// Return if no parameter is remaining...
IF ( ParameterCnt = 0 ) THEN RETURN; END_IF
// dec remaining parameter(s)                        
ParameterCnt := ParameterCnt - 1;
// Create log entry for HoldToRun
CreateLogMessagePara1 ( Timestamp   := AxesGroup.State.SystemTime,
                        MessageType := MessageType.CMD,
                        Severity    := Severity.DEBUG,
                        MessageCode := 0,
                        MessageText := 'Command.HoldToRun = {1}',
                        Para1       :=  BOOL_TO_STRING(_command.HoldToRun));
                        

// Return if no parameter is remaining...
IF ( ParameterCnt = 0 ) THEN RETURN; END_IF
// dec remaining parameter(s)                        
ParameterCnt := ParameterCnt - 1;
// Create log entry for StepMode
CreateLogMessagePara1 ( Timestamp   := AxesGroup.State.SystemTime,
                        MessageType := MessageType.CMD,
                        Severity    := Severity.DEBUG,
                        MessageCode := 0,
                        MessageText := 'Command.StepMode = {1}',
                        Para1       :=  USINT_TO_STRING(_command.StepMode));
                                                

// Return if no parameter is remaining...
IF ( ParameterCnt = 0 ) THEN RETURN; END_IF
// dec remaining parameter(s)                        
ParameterCnt := ParameterCnt - 1;
// Create log entry for ManualStep
CreateLogMessagePara1 ( Timestamp   := AxesGroup.State.SystemTime,
                        MessageType := MessageType.CMD,
                        Severity    := Severity.DEBUG,
                        MessageCode := 0,
                        MessageText := 'Command.ManualStep = {1}',
                        Para1       :=  BOOL_TO_STRING(_command.ManualStep));

                
END_METHOD

METHOD FB_init : BOOL
VAR_INPUT
  /// if TRUE, the retain variables are initialized (warm start / cold start)
  bInitRetains : BOOL; 
  /// if TRUE, the instance afterwards gets moved into the copy code (online change)
  bInCopyCode  : BOOL;  
END_VAR
                  MyType := 'MC_EnableRobotFB';

ExecMode := ExecutionMode.PARALLEL;
Priority := PriorityLevel.NORMAL;
                
END_METHOD

METHOD Protected OnExecCancel : DINT
VAR_IN_OUT
  /// Robot assignment of function
  AxesGroup : AxesGroup; 
END_VAR
VAR
  /// internal return value 
 _retVal    : DINT;
END_VAR
                  OnExecCancel := RobotLibraryConstants.RUNNING;

CASE _stepCancel OF
  
  0: // set busy flag
     Busy := TRUE;
    
     // Create log entry
     CreateLogMessagePara1 ( Timestamp   := AxesGroup.State.SystemTime,
                             MessageType := MessageType.CMD,
                             Severity    := Severity.DEBUG,
                             MessageCode := 0,
                             MessageText := 'Execution of {1} cancelled',
                             Para1       := MyType);                 
    
     // try to remove cmd
    _retVal := AxesGroup.Acyclic.ActiveCommandRegister.RemoveCmd(_uniqueID);
  
     // check result of removement       
     IF ( _retVal = RobotLibraryConstants.OK )
     THEN
       // Reset step counter
      _stepCancel := 0;
       // finished okay
       OnExecCancel := RobotLibraryConstants.OK;
     
       // Create log entry
       CreateLogMessagePara1 ( Timestamp   := AxesGroup.State.SystemTime,
                               MessageType := MessageType.CMD,
                               Severity    := Severity.DEBUG,
                               MessageCode := 0,
                               MessageText := '{1} successfully removed from ACR',
                               Para1       := MyType);                 
     ELSE
       // set timeout
       SetTimeout(PT := _timeoutCancel, rTimer := _timerCancel);
       // inc step counter
      _stepCancel := _stepCancel + 1; 
     
       // Create log entry
       CreateLogMessagePara1 ( Timestamp   := AxesGroup.State.SystemTime,
                               MessageType := MessageType.CMD,
                               Severity    := Severity.DEBUG,
                               MessageCode := 0,
                               MessageText := '{1} was not removed from ACR because execution was already in progress',
                               Para1       := MyType);                 
     END_IF       
  
     
 1:  // call clear error 
     OnExecCancel := OnExecErrorClear(AxesGroup := AxesGroup);  
 
     IF ( OnExecCancel = RobotLibraryConstants.OK)
     THEN
       // Reset busy flag
       Busy := FALSE;
       // Reset step counter
      _stepCancel := 0;
       // finished okay
       OnExecCancel := RobotLibraryConstants.OK;
     END_IF  
  
ELSE
  // invalid step
  SetError( ErrorID := RobotLibraryErrorIdEnum.ERR_INVALID_STEP, Overwrite := TRUE );
END_CASE  


                        
// reset step counter
IF (OnExecCancel <> RobotLibraryConstants.RUNNING)
THEN
  // Reset FB variables
  Reset();
  // Reset step counter
 _stepCancel := 0;
END_IF                        
                
END_METHOD

METHOD PROTECTED OnExecErrorClear : DINT
VAR_IN_OUT
  /// Robot assignment of function
  AxesGroup : AxesGroup; 
END_VAR
                  OnExecErrorClear := RobotLibraryConstants.RUNNING;

CASE _stepClearError OF
  
  0:  // set busy flag
      Busy := TRUE;
      // trigger parameter update to disable FB
     _parameterUpdateInternal := TRUE;
      // call Check Parameter changed method to trigger the parameter update to disable the function
      CheckParameterChanged(AxesGroup := AxesGroup);
      // set timeout
      SetTimeout(PT := _timeoutClearError, rTimer := _timerClearError);
      // inc step counter
     _stepClearError := _stepClearError + 1; 
      
  1: IF ( _responseReceived )
     THEN
       // reset response received flag
      _responseReceived := FALSE;
       // reset step counter
      _stepClearError := 0;
       // finished
       OnExecErrorClear := RobotLibraryConstants.OK;
     ELSE
       // timeout exceeded ? 
       IF (CheckTimeout(_timerClearError) = RobotLibraryConstants.OK)
       THEN
         OnExecErrorClear := RobotLibraryConstants.HAS_ERROR;
       END_IF
	   END_IF
ELSE
  // invalid step
  SetError( ErrorID := RobotLibraryErrorIdEnum.ERR_INVALID_STEP, Overwrite := TRUE );
END_CASE


// reset step counter
IF (OnExecErrorClear <> RobotLibraryConstants.RUNNING)
THEN
  // Reset 
  Reset();     
  // reset step counter
 _stepClearError := 0;
END_IF
                
END_METHOD

METHOD PROTECTED OnExecRun : DINT
VAR_IN_OUT
  /// Robot assignment of function
  AxesGroup : AxesGroup; 
END_VAR
                  SUPER^.OnExecRun(AxesGroup := AxesGroup);

CASE _stepCmd OF
  
  00:  IF ( _enable_R.Q ) AND ( NOT Error) 
       THEN
         // reset the rising edge
        _enable_R();       

         // Check function is supported and parameter are valid ?
         IF (( CheckFunctionSupported   ( AxesGroup := AxesGroup )) AND
             ( CheckParameterValid      ( AxesGroup := AxesGroup )) AND
             ( CheckSynchronizationValid( AxesGroup := AxesGroup )))      
         THEN
           // Reset all internal flags
           Reset();
           // set busy flag
           Busy := TRUE;
           // Reset command outputs
           SysDepMemSet(pDest := ADR(OutCmd), Value := 0, DataLen := SIZEOF(OutCmd));         
           // apply command parameter
          _parCmd := ParCmd;
           // init parameter sequence
          _command.ParSeq := 1;
           // create command data
           CommandData := CreateCommandPayload(AxesGroup := AxesGroup);
           // Add command to active command register
          _uniqueID := AxesGroup.Acyclic.ActiveCommandRegister.AddCmd( pCommandFB := ADR(THIS^ ));     
           // set timeout
           SetTimeout(PT := _timeoutCmd, rTimer := _timerCmd);
           // inc step counter
          _stepCmd := _stepCmd + 1; 
         END_IF
       END_IF
     

  01:  // Wait for responce received
       IF ( _responseReceived )
       THEN
         // reset response received flag
        _responseReceived := FALSE;
         // update state flags
         OnUpdateStateFlags(_response.State);
         // update state flags
         OnApplyOutCmd(_response.State);
       END_IF
       
       // do not abort directly, so that the ParSeq update can be send
       IF ( _enable_F.Q ) 
       THEN
         // Set Busy flag
         Busy := TRUE;
         // trigger parameter update to disable FB
        _parameterUpdateInternal := TRUE;        
         // reset the falling edge
        _enable_F();
         // set timeout
         SetTimeout(PT := _timeoutCmd, rTimer := _timerCmd);
         // inc step counter
        _stepCmd := _stepCmd + 1; 
       END_IF

      // Wait for response received or timeout or not Initialized
  02: IF ((    _responseReceived                                   )  OR 
          (     CheckTimeout(_timerCmd) = RobotLibraryConstants.OK )) OR 
         (( NOT AxesGroup.State.Initialized                        )  AND
          ( NOT AxesGroup.State.Synchronized                       ))
      THEN
        Reset();   
	    END_IF
      
ELSE
  // invalid step
  SetError( ErrorID := RobotLibraryErrorIdEnum.ERR_INVALID_STEP, Overwrite := TRUE );
END_CASE



// Reset FB
IF (( _enable_R.Q ) OR
    ( _enable_F.Q ))
THEN
  Reset();
END_IF
                
END_METHOD

METHOD PROTECTED OnUpdateStateFlags
VAR_INPUT
  /// Command message state
  State : CmdMessageState;
END_VAR
                  // Reset State flags
;

// Update results
Enabled := _response.Enabled;

CASE State OF

  // No operation or process is active
  CmdMessageState.EMPTY               :;
  // Created but not yet started
  CmdMessageState.CREATED             :;
  // Buffered and awaiting execution
  CmdMessageState.BUFFERED            : CommandBuffered    := TRUE;
                                        ParameterAccepted  := TRUE;  
  // Buffered in planner for future execution
  CmdMessageState.BUFFERED_IN_PLANNER : CommandBuffered    := TRUE;
                                        ParameterAccepted  := TRUE;
  // Currently active and in progress
  CmdMessageState.ACTIVE              : IF (Enabled = Enable)
                                        THEN  
                                          Busy := FALSE;   
                                        END_IF
                                       
  // Interrupted and awaiting continuation
  CmdMessageState.INTERRUPTED         :;  
  // Requested for abort
  CmdMessageState.ABORT_REQUEST       :;
  // Successfully completed
  CmdMessageState.DONE                : Busy               := FALSE;
  // Aborted before completion
  CmdMessageState.ABORTED             : Busy               := FALSE;
  // Encountered an error during execution
  CmdMessageState.ERROR               : Error              := TRUE;
                                        Busy               := FALSE;
END_CASE
                
END_METHOD

METHOD INTERNAL ParseResponsePayload : DINT
VAR_INPUT
  /// Response data
  ResponseData : RobotLibraryResponseDataFB;
  /// Timestamp
  Timestamp    : SystemTime;  
END_VAR
VAR
  /// Parameter count
 _parameterCnt : DINT;
END_VAR
// Table 6-26: Received CMD payload (RC to PLC) of "EnableRobot"
// --------------------------
// Header
// --------------------------
// Byte 00 : USINT - ParSeq | State     
// Byte 01 : SINT  - AlarmMessageSeverity    
// Byte 02 : UINT  - AlarmMessageCode HB
// Byte 03 :       - AlarmMessageCode LB
// --------------------------
// Datablock
// --------------------------
// Byte 04 : BOOL  - Enabled
// --------------------------
                  // call base implementation to parse the header from payload buffer
ResponseData.PayloadPtr := SUPER^.ParseResponsePayload(ResponseData := ResponseData, Timestamp := Timestamp);

// copy parsed header to response
_response.ParSeq               := _rspHeader.ParSeq;
_response.State                := _rspHeader.State;
_response.AlarmMessageSeverity := _rspHeader.AlarmMessageSeverity;
_response.AlarmMessageCode     := _rspHeader.AlarmMessageCode;


// Check payload remaining ? 
IF ( ResponseData.IsPayloadRemaining)
THEN 
  // Get Response.Enabled
 _response.Enabled := ResponseData.GetBool();
  // inc parameter counter
 _parameterCnt := _parameterCnt + 1;
END_IF


// Create logging
ParseResponsePayloadLog(ResponseData := ResponseData, Timestamp := Timestamp, ParameterCnt := _parameterCnt);
                
END_METHOD

METHOD INTERNAL ParseResponsePayloadLog
VAR_INPUT
  /// Response data
  ResponseData : RobotLibraryResponseDataFB;
  /// Timestamp
  Timestamp    : SystemTime;  
  /// Parameter count
  ParameterCnt : DINT;
END_VAR
                  // Create log entry for Parameter start
CreateLogMessagePara1 ( Timestamp   := Timestamp,
                        MessageType := MessageType.CMD,
                        Severity    := Severity.DEBUG,
                        MessageCode := 0,
                        MessageText := '{1} parameter(s) to parse from the response data:',
                        Para1       := DINT_TO_STRING(ParameterCnt));
                        
// Return if no parameter is remaining...
IF ( ParameterCnt = 0 ) THEN RETURN; END_IF
// dec remaining parameter(s)                        
ParameterCnt := ParameterCnt - 1;

// Create log entry for Enabled
CreateLogMessagePara1 ( Timestamp   := Timestamp,
                        MessageType := MessageType.CMD,
                        Severity    := Severity.DEBUG,
                        MessageCode := 0,
                        MessageText := 'Response.Enabled = {1}',
                        Para1       :=  BOOL_TO_STRING(_response.Enabled));


                
END_METHOD

METHOD PROTECTED Reset : DINT
VAR_INPUT
END_VAR
                  SUPER^.Reset();

Busy               := FALSE;
CommandBuffered    := FALSE;
ParameterAccepted  := FALSE;
                
END_METHOD
END_FUNCTION_BLOCK

/// Acknowledgement all pending errors
FUNCTION_BLOCK MC_GroupResetFB EXTENDS RobotLibraryBaseExecuteFB
// ------------------------------------------------------------------------- 
//  SRCI Robot Library                                                
// ------------------------------------------------------------------------- 
//                                                                           
//  Object:      GroupResetFB                                       
//  Author:      Thorsten Brach                                                
//  Date:        2024-06-01
//
//  Description:                                              
//   
//                                                                           
//  Copyright: 
//    (C) 2024 Thorsten Brach. All rights reserved                                                                                                                                            
//             Licensed under the MIT License.
//                                                                           
//  Disclaimer:                                                                           
//    This project is provided without any guarantee and can be used for   
//    private and commercial purposes. Any use is at the user’s 
//    own risk and responsibility.
//
// -------------------------------------------------------------------------
VAR_INPUT
  /// Command parameter 
  ParCmd          : GroupResetParCmd;      
END_VAR

VAR_OUTPUT
  /// Command output 
  OutCmd          : GroupResetOutCmd;   
  /// Command is transferred and confirmed by the RC
  CommandBuffered : BOOL;     
END_VAR
VAR
  /// internal copy of command parameter 
 _parCmd          : GroupResetParCmd;
  /// command data to send
 _command         : GroupResetSendData;
  /// response data received
 _response        : GroupResetRecvData;      
END_VAR

            SUPER^(AxesGroup := AxesGroup);
          

METHOD INTERNAL CheckAddParameter : BOOL
VAR_INPUT
  /// Payload pointer
  PayloadPtr : UDINT;
END_VAR
VAR
  /// Payload as byte array
  Payload    : ARRAY [1..SIZEOF(_command)] OF BYTE;
  /// Null Byte array 
  Null       : ARRAY [1..SIZEOF(_command)] OF BYTE;
  /// Data length to compare
  DataLen    : UDINT;
END_VAR
                  // Payload pointer must be decreased by one byte, because ADR(Payload) is already one byte !
PayloadPtr := LIMIT (0, PayloadPtr - 1, SIZEOF(Payload) -1);
// Convert command struct to payload array
SysDepMemCpy( pDest := ADR(Payload), pSrc := ADR(_command), DataLen := SIZEOF(_command));
// Calculate the data length to compare - at least one byte must be compared !
DataLen := LIMIT(1, SIZEOF(Payload) - PayloadPtr, SIZEOF(Payload)); 
// Compare Payload-Array with Null-Byte-Array
CheckAddParameter := SysDepMemCmp( pData1 := ADR(Payload) + PayloadPtr , pData2 := ADR(Null), DataLen := DataLen) <>  RobotLibraryConstants.OK ;
                
END_METHOD

METHOD PROTECTED CheckFunctionSupported : BOOL
VAR_IN_OUT
  /// Robot assignment of function
  AxesGroup : AxesGroup; 
END_VAR
                  CheckFunctionSupported := AxesGroup.State.RobotData.RCSupportedFunctions.GroupReset;

IF ( NOT CheckFunctionSupported )
THEN
  // call base implementation for set error and create log entry
  SUPER^.CheckFunctionSupported(AxesGroup := AxesGroup);
END_IF
                
END_METHOD

METHOD PROTECTED CheckParameterChanged : BOOL
VAR_IN_OUT
  /// Robot assignment of function
  AxesGroup    : AxesGroup; 
END_VAR
                  IF (SIZEOF(ParCmd) = 0) OR (_stepCmd = 0)
THEN
  RETURN;
END_IF
 
// compare memory
_parameterChanged := ( SysDepMemCmp(pData1 := ADR(ParCmd), pData2 := ADR(_parCmd), DataLen := SIZEOF(ParCmd)) <> RobotLibraryConstants.OK );

// check parameter valid ?
_parameterValid   := CheckParameterValid( AxesGroup := AxesGroup );

IF ((  _parameterChanged        )  AND 
    (  _parameterValid          )) OR
    (  _parameterUpdateInternal )  
THEN  
  // Create log entry for parameter changed event
  CreateLogMessagePara1 ( Timestamp   := AxesGroup.State.SystemTime,
                          MessageType := MessageType.CMD,
                          Severity    := Severity.DEBUG,
                          MessageCode := 0,
                          MessageText := 'NotifyParameterChanged Event {1}',
                          Para1       :=  '' );

  // reset internal flag for send parameter update
 _parameterUpdateInternal := FALSE;
  // update internal copy of parameters 
 _parCmd := ParCmd;
  // inc parameter sequence
 _command.ParSeq := _command.ParSeq + 1;
  // update command data  
  CommandData := CreateCommandPayload(AxesGroup := AxesGroup); // ( Access via reference to rCommandFB in ACR )
  // notify active command register 
  AxesGroup.Acyclic.ActiveCommandRegister.NotifyParameterChanged := _uniqueID;
END_IF
                
END_METHOD

METHOD INTERNAL CreateCommandPayload : RobotLibraryCommandDataFB
VAR_IN_OUT
  /// Robot assignment of function
  AxesGroup : AxesGroup; 
END_VAR
VAR
  /// Parameter count
 _parameterCnt : DINT;
END_VAR
// Table 6-31: Sent CMD payload (PLC to RC) of "GroupReset"
// --------------------------
// Header
// --------------------------
// Byte 00 : UINT  - Type HB     
// Byte 01 :       - Type LB    
// Byte 02 : USINT - Reserve | ExecutionMode
// Byte 03 : USINT - ParSeq  | Priority
// --------------------------
                  // set command parameter 
_command.CmdTyp     :=  CmdType.GroupReset;
_command.ExecMode   :=  ExecMode;
_command.ParSeq     := _command.ParSeq;
_command.Priority   :=  Priority;

// copy command data to header
_cmdHeader := _command;
// call base implementation to copy header to payload buffer
CreateCommandPayload := SUPER^.CreateCommandPayload(AxesGroup := AxesGroup);


// Create logging
CreateCommandPayloadLog(AxesGroup := AxesGroup, ParameterCnt := _parameterCnt);
                
END_METHOD

METHOD INTERNAL CreateCommandPayloadLog
VAR_IN_OUT
  /// Robot assignment of function
  AxesGroup : AxesGroup; 
END_VAR
VAR_INPUT
  /// Parameter count
  ParameterCnt : DINT;
END_VAR
                  // Create log entry for Parameter start
CreateLogMessagePara1 ( Timestamp   := AxesGroup.State.SystemTime,
                        MessageType := MessageType.CMD,
                        Severity    := Severity.DEBUG,
                        MessageCode := 0,
                        MessageText := 'Create command payload with {1} parameter(s) :',
                        Para1       := DINT_TO_STRING(ParameterCnt));
                
END_METHOD

METHOD FB_init : BOOL
VAR_INPUT
  /// if TRUE, the retain variables are initialized (warm start / cold start)
  bInitRetains : BOOL; 
  /// if TRUE, the instance afterwards gets moved into the copy code (online change)
  bInCopyCode  : BOOL;  
END_VAR
                  MyType := 'MC_GroupResetFB';

ExecMode := ExecutionMode.PARALLEL;
Priority := PriorityLevel.NORMAL;
                
END_METHOD

METHOD PROTECTED OnExecRun : DINT
VAR_IN_OUT
  /// Robot assignment of function
  AxesGroup : AxesGroup; 
END_VAR
                  // call base implementation
SUPER^.OnExecRun(AxesGroup := AxesGroup);

CASE _stepCmd OF
  
  00:  IF ( _execute_R.Q ) AND ( NOT Error)
       THEN
         IF (( CheckFunctionSupported( AxesGroup := AxesGroup )) AND
             ( CheckParameterValid   ( AxesGroup := AxesGroup )))      
         THEN
           // set busy flag
           Busy := TRUE;
           // Reset command outputs
           SysDepMemSet(pDest := ADR(OutCmd), Value := 0, DataLen := SIZEOF(OutCmd));         
           // apply command parameter
          _parCmd := ParCmd;
           // init parameter sequence
          _command.ParSeq := 1;
           // create command data
           CommandData := CreateCommandPayload(AxesGroup := AxesGroup);
           // Add command to active command register
          _uniqueID := AxesGroup.Acyclic.ActiveCommandRegister.AddCmd( pCommandFB := ADR(THIS^ ));     
           // set timeout
           SetTimeout(PT := _timeoutCmd, rTimer := _timerCmd);
           // inc step counter
          _stepCmd := _stepCmd + 1;
         END_IF 
       END_IF
     

  01:  // Wait for responce received
       IF ( _responseReceived )
       THEN
         // reset response received flag
        _responseReceived := FALSE;
         // update state flags
         OnUpdateStateFlags(_response.State);
         // update state flags
         OnApplyOutCmd(_response.State);
               
         // Done, Aborted or Error ?
         IF (_response.State >= CmdMessageState.DONE )
         THEN
           // Reset FastStop counter
           AxesGroup.Cyclic.PlcToRob.FastStop := 0; 
           // set timeout
           SetTimeout(PT := _timeoutCmd, rTimer := _timerCmd);
           // inc step counter
          _stepCmd := _stepCmd + 1; 
         END_IF
       END_IF


  02: IF ( NOT Execute)
      THEN
        Reset();
      END_IF     

ELSE
  // invalid step
  SetError( ErrorID := RobotLibraryErrorIdEnum.ERR_INVALID_STEP, Overwrite := TRUE );
END_CASE


// Reset FB
IF ( NOT Execute )
THEN
  Reset();
END_IF

// forwarding GroupReset Info
AxesGroup.State.GroupReset := Execute;
                
END_METHOD

METHOD PROTECTED OnUpdateStateFlags
VAR_INPUT
  /// Command message state
  State : CmdMessageState;
END_VAR
                  // Reset State flags
Done := FALSE;

CASE State OF

  // No operation or process is active
  CmdMessageState.EMPTY               :;
  // Created but not yet started
  CmdMessageState.CREATED             :;
  // Buffered and awaiting execution
  CmdMessageState.BUFFERED            : CommandBuffered    := TRUE;
  // Buffered in planner for future execution
  CmdMessageState.BUFFERED_IN_PLANNER : CommandBuffered    := TRUE;
  // Currently active and in progress
  CmdMessageState.ACTIVE              :;                                         
  // Interrupted and awaiting continuation
  CmdMessageState.INTERRUPTED         :;  
  // Requested for abort
  CmdMessageState.ABORT_REQUEST       :;
  // Successfully completed
  CmdMessageState.DONE                : Done               := TRUE;
                                        Busy               := FALSE;
  // Aborted before completion
  CmdMessageState.ABORTED             : Busy               := FALSE;
  // Encountered an error during execution
  CmdMessageState.ERROR               : Error              := TRUE;
                                        Busy               := FALSE;
END_CASE
                
END_METHOD

METHOD INTERNAL ParseResponsePayload : DINT
VAR_INPUT
  /// Response data
  ResponseData : RobotLibraryResponseDataFB;
  /// Timestamp
  Timestamp    : SystemTime;  
END_VAR
VAR
  /// Parameter count
 _parameterCnt : DINT;
END_VAR
// Table 6-32: Received CMD payload (RC to PLC) of "GroupReset"
// --------------------------
// Header
// --------------------------
// Byte 00 : USINT - ParSeq | State     
// Byte 01 : SINT  - AlarmMessageSeverity    
// Byte 02 : UINT  - AlarmMessageCode HB
// Byte 03 :       - AlarmMessageCode LB
                  // call base implementation to parse the header from payload buffer
ResponseData.PayloadPtr := SUPER^.ParseResponsePayload(ResponseData := ResponseData, Timestamp := Timestamp);

// copy parsed header to response
_response.ParSeq               := _rspHeader.ParSeq;
_response.State                := _rspHeader.State;
_response.AlarmMessageSeverity := _rspHeader.AlarmMessageSeverity;
_response.AlarmMessageCode     := _rspHeader.AlarmMessageCode;

// Create logging
ParseResponsePayloadLog(ResponseData := ResponseData, Timestamp := Timestamp, ParameterCnt := _parameterCnt);
                
END_METHOD

METHOD INTERNAL ParseResponsePayloadLog
VAR_INPUT
  /// Response data
  ResponseData : RobotLibraryResponseDataFB;
  /// Timestamp
  Timestamp    : SystemTime;  
  /// Parameter count
  ParameterCnt : DINT;
END_VAR
                  // Create log entry for Parameter start
CreateLogMessagePara1 ( Timestamp   := Timestamp,
                        MessageType := MessageType.CMD,
                        Severity    := Severity.DEBUG,
                        MessageCode := 0,
                        MessageText := '{1} parameter(s) to parse from the response data:',
                        Para1       := DINT_TO_STRING(ParameterCnt));
                        

// Return if no parameter is remaining...
IF ( ParameterCnt = 0 ) THEN RETURN; END_IF
// dec remaining parameter(s)                        
ParameterCnt := ParameterCnt - 1;
// Create log entry for no parameter 
CreateLogMessage      ( Timestamp   := Timestamp,
                        MessageType := MessageType.CMD,
                        Severity    := Severity.DEBUG,
                        MessageCode := 0,
                        MessageText := 'This command has no parameter to parse...');
                
END_METHOD

METHOD PROTECTED Reset : DINT
VAR_INPUT
END_VAR
                  Reset := SUPER^.Reset();

Done               := FALSE;
Busy               := FALSE;
CommandBuffered    := FALSE;


                
END_METHOD
END_FUNCTION_BLOCK

FUNCTION_BLOCK MC_ReadServerLog EXTENDS RobotLibraryBaseFB
VAR
END_VAR

            
          

METHOD FB_init : BOOL
VAR_INPUT
  /// if TRUE, the retain variables are initialized (warm start / cold start)
  bInitRetains : BOOL; 
  /// if TRUE, the instance afterwards gets moved into the copy code (online change)
  bInCopyCode  : BOOL;  
END_VAR
                  MyType := 'MC_ReadServerLogFB';

ExecMode := ExecutionMode.PARALLEL;
Priority := PriorityLevel.NORMAL;
                
END_METHOD
END_FUNCTION_BLOCK

/// Restart/reboot of the RC.
FUNCTION_BLOCK MC_RestartControllerFB EXTENDS RobotLibraryBaseExecuteFB
// ------------------------------------------------------------------------- 
//  SRCI Robot Library                                                
// ------------------------------------------------------------------------- 
//                                                                           
//  Object:      RestartControllerFB                                       
//  Author:      Thorsten Brach                                                
//  Date:        2024-06-01
//
//  Description:                                              
//   
//                                                                           
//  Copyright: 
//    (C) 2024 Thorsten Brach. All rights reserved                                                                                                                                            
//             Licensed under the MIT License.
//                                                                           
//  Disclaimer:                                                                           
//    This project is provided without any guarantee and can be used for   
//    private and commercial purposes. Any use is at the user’s 
//    own risk and responsibility.
//
// -------------------------------------------------------------------------
VAR_INPUT
  /// Command parameter 
  ParCmd          : RestartControllerParCmd;  
END_VAR

VAR_OUTPUT
  /// Command is transferred and confirmed by the RC
  CommandBuffered : BOOL;
  /// Command outputs 
  OutCmd          : RestartControllerOutCmd;  
END_VAR

VAR
  /// internal copy of command parameter 
 _parCmd          : RestartControllerParCmd;
  /// command data to send
 _command         : RestartControllerSendData;
  /// response data received
 _response        : RestartControllerRecvData;      
END_VAR

            SUPER^(AxesGroup := AxesGroup);
          

METHOD INTERNAL CheckAddParameter : BOOL
VAR_INPUT
  /// Payload pointer
  PayloadPtr : UDINT;
END_VAR
VAR
  /// Payload as byte array
  Payload    : ARRAY [1..SIZEOF(_command)] OF BYTE;
  /// Null Byte array 
  Null       : ARRAY [1..SIZEOF(_command)] OF BYTE;
  /// Data length to compare
  DataLen    : UDINT;
END_VAR
                  // Payload pointer must be decreased by one byte, because ADR(Payload) is already one byte !
PayloadPtr := LIMIT (0, PayloadPtr - 1, SIZEOF(Payload) -1);
// Convert command struct to payload array
SysDepMemCpy( pDest := ADR(Payload), pSrc := ADR(_command), DataLen := SIZEOF(_command));
// Calculate the data length to compare - at least one byte must be compared !
DataLen := LIMIT(1, SIZEOF(Payload) - PayloadPtr, SIZEOF(Payload)); 
// Compare Payload-Array with Null-Byte-Array
CheckAddParameter := SysDepMemCmp( pData1 := ADR(Payload) + PayloadPtr , pData2 := ADR(Null), DataLen := DataLen) <>  RobotLibraryConstants.OK ;
                
END_METHOD

METHOD PROTECTED CheckFunctionSupported : BOOL
VAR_IN_OUT
  /// Robot assignment of function
  AxesGroup : AxesGroup; 
END_VAR
                  CheckFunctionSupported := AxesGroup.State.RobotData.RCSupportedFunctions.RestartController;

IF ( NOT CheckFunctionSupported )
THEN
  // call base implementation for set error and create log entry
  SUPER^.CheckFunctionSupported(AxesGroup := AxesGroup);
END_IF
                
END_METHOD

METHOD PROTECTED CheckParameterChanged : BOOL
VAR_IN_OUT
  /// Robot assignment of function
  AxesGroup    : AxesGroup; 
END_VAR
                  // Check ParCmd Size is > 0, because MemCmp does not work correctly with size = 0
IF (SIZEOF(ParCmd) = 0) OR (_stepCmd = 0)
THEN 
  RETURN;
END_IF

// compare memory 
_parameterChanged := ( SysDepMemCmp(pData1 := ADR(ParCmd), pData2 := ADR(_parCmd), DataLen := SIZEOF(ParCmd)) <> RobotLibraryConstants.OK );

// check parameter valid ?
_parameterValid   := CheckParameterValid( AxesGroup := AxesGroup );

IF ((  _parameterChanged        )  AND 
    (  _parameterValid          )) OR
    (  _parameterUpdateInternal )  
THEN  
  // Create log entry for parameter changed event
  CreateLogMessagePara1 ( Timestamp   := AxesGroup.State.SystemTime,
                          MessageType := MessageType.CMD,
                          Severity    := Severity.DEBUG,
                          MessageCode := 0,
                          MessageText := 'NotifyParameterChanged Event {1}',
                          Para1       :=  '' );

  // reset internal flag for send parameter update
 _parameterUpdateInternal := FALSE;
  // update internal copy of parameters 
 _parCmd := ParCmd;
  // inc parameter sequence
 _command.ParSeq := _command.ParSeq + 1;
  // update command data  
  CommandData := CreateCommandPayload(AxesGroup := AxesGroup); // ( Access via reference to rCommandFB in ACR )
  // notify active command register 
  AxesGroup.Acyclic.ActiveCommandRegister.NotifyParameterChanged := _uniqueID;
END_IF
                
END_METHOD

METHOD INTERNAL CreateCommandPayload : RobotLibraryCommandDataFB
VAR_IN_OUT
  /// Robot assignment of function
  AxesGroup : AxesGroup; 
END_VAR
VAR
  /// Parameter count
 _parameterCnt : DINT;
END_VAR
// Table 6-57: Sent CMD payload (PLC to RC) of "RestartController"
// --------------------------
// Header
// --------------------------
// Byte 00 : UINT  - Type HB     
// Byte 01 :       - Type LB    
// Byte 02 : USINT - Reserve | ExecutionMode
// Byte 03 : USINT - ParSeq  | Priority
// --------------------------
                  // set command parameter 
_command.CmdTyp     :=  CmdType.RestartController;
_command.ExecMode   :=  ExecMode;
_command.ParSeq     := _command.ParSeq;
_command.Priority   :=  Priority;


// copy command data to header
_cmdHeader := _command;
// call base implementation to copy header to payload buffer
CreateCommandPayload := SUPER^.CreateCommandPayload(AxesGroup := AxesGroup);


// Create logging
CreateCommandPayloadLog(AxesGroup := AxesGroup, ParameterCnt := _parameterCnt);
                
END_METHOD

METHOD INTERNAL CreateCommandPayloadLog
VAR_IN_OUT
  /// Robot assignment of function
  AxesGroup : AxesGroup; 
END_VAR
VAR_INPUT
  /// Parameter count
  ParameterCnt : DINT;
END_VAR
                  // Create log entry for Parameter start
CreateLogMessagePara1 ( Timestamp   := AxesGroup.State.SystemTime,
                        MessageType := MessageType.CMD,
                        Severity    := Severity.DEBUG,
                        MessageCode := 0,
                        MessageText := 'Create command payload with {1} parameter(s) :',
                        Para1       := DINT_TO_STRING(ParameterCnt));
                
END_METHOD

METHOD FB_init : BOOL
VAR_INPUT
  /// if TRUE, the retain variables are initialized (warm start / cold start)
  bInitRetains : BOOL; 
  /// if TRUE, the instance afterwards gets moved into the copy code (online change)
  bInCopyCode  : BOOL;  
END_VAR
                  MyType := 'MC_RestartControllerFB';

ExecMode := ExecutionMode.PARALLEL;
Priority := PriorityLevel.NORMAL;
                
END_METHOD

METHOD PROTECTED OnApplyOutCmd
VAR_INPUT
  /// Command message state
  State : CmdMessageState;
END_VAR
                  IF ( State = CmdMessageState.EMPTY ) 
THEN
  // Reset command outputs
  SysDepMemSet(pDest := ADR(OutCmd), Value := 0, DataLen := SIZEOF(OutCmd));         
END_IF

IF (( State = CmdMessageState.ACTIVE ) OR
    ( State = CmdMessageState.DONE   ))
THEN
  // Update results
  OutCmd.RestartAccepted := _response.RestartAccepted;
END_IF
                
END_METHOD

METHOD PROTECTED OnExecRun : DINT
VAR_IN_OUT
  /// Robot assignment of function
  AxesGroup : AxesGroup; 
END_VAR
                  // call base implementation
SUPER^.OnExecRun(AxesGroup := AxesGroup);

CASE _stepCmd OF
  
  00:  IF ( _execute_R.Q ) AND ( NOT Error)   
       THEN
         // Check function is supported and parameter are valid ?
         IF (( CheckFunctionSupported( AxesGroup := AxesGroup )) AND
             ( CheckParameterValid   ( AxesGroup := AxesGroup )))      
         THEN
           // set busy flag
           Busy := TRUE;
           // Reset command outputs
           SysDepMemSet(pDest := ADR(OutCmd), Value := 0, DataLen := SIZEOF(OutCmd));         
           // apply command parameter
          _parCmd := ParCmd;
           // init parameter sequence
          _command.ParSeq := 1;
           // create command data
           CommandData := CreateCommandPayload(AxesGroup := AxesGroup);
           // Add command to active command register
          _uniqueID := AxesGroup.Acyclic.ActiveCommandRegister.AddCmd( pCommandFB := ADR(THIS^ ));     
           // set timeout
           SetTimeout(PT := _timeoutCmd, rTimer := _timerCmd);
           // inc step counter
          _stepCmd := _stepCmd + 1;
         END_IF 
       END_IF
     

  01:  // Wait for responce received
       IF ( _responseReceived )
       THEN
         // reset response received flag
        _responseReceived := FALSE;
         // update state flags
         OnUpdateStateFlags(_response.State);
         // update state flags
         OnApplyOutCmd(_response.State);

         // Done, Aborted or Error ?
         IF (_response.State >= CmdMessageState.DONE )
         THEN
           // set timeout
           SetTimeout(PT := _timeoutCmd, rTimer := _timerCmd);
           // inc step counter
          _stepCmd := _stepCmd + 1; 
         END_IF
       END_IF


  02: IF ( NOT Execute)
      THEN
        Reset();
      END_IF     

ELSE
  // invalid step
  SetError( ErrorID := RobotLibraryErrorIdEnum.ERR_INVALID_STEP, Overwrite := TRUE );
END_CASE


// Reset FB
IF ( NOT Execute )
THEN
  Reset();
END_IF
                
END_METHOD

METHOD PROTECTED OnUpdateStateFlags
VAR_INPUT
  /// Command message state
  State : CmdMessageState;
END_VAR
                  // Reset State flags
Done := FALSE;

CASE State OF

  // No operation or process is active
  CmdMessageState.EMPTY               :;
  // Created but not yet started
  CmdMessageState.CREATED             :;
  // Buffered and awaiting execution
  CmdMessageState.BUFFERED            : CommandBuffered    := TRUE;
  // Buffered in planner for future execution
  CmdMessageState.BUFFERED_IN_PLANNER : CommandBuffered    := TRUE;
  // Currently active and in progress
  CmdMessageState.ACTIVE              :;
  // Interrupted and awaiting continuation
  CmdMessageState.INTERRUPTED         :;  
  // Requested for abort
  CmdMessageState.ABORT_REQUEST       :;
  // Successfully completed
  CmdMessageState.DONE                : Done               := TRUE;
                                        Busy               := FALSE;
  // Aborted before completion
  CmdMessageState.ABORTED             : Busy               := FALSE;
  // Encountered an error during execution
  CmdMessageState.ERROR               : Error              := TRUE;
                                        Busy               := FALSE;
END_CASE
                
END_METHOD

METHOD INTERNAL ParseResponsePayload : DINT
VAR_INPUT
  /// Response data
  ResponseData : RobotLibraryResponseDataFB;
  /// Timestamp
  Timestamp    : SystemTime;  
END_VAR
VAR
  /// Parameter count
 _parameterCnt : DINT;
END_VAR
// Table 6-58: Received CMD payload (RC to PLC) of "RestartController"
// --------------------------
// Header
// --------------------------
// Byte 00 : USINT - ParSeq | State     
// Byte 01 : SINT  - AlarmMessageSeverity    
// Byte 02 : UINT  - AlarmMessageCode HB
// Byte 03 :       - AlarmMessageCode LB
// --------------------------
// Datablock
// --------------------------
// Byte 4  : BOOL  - RestartAccepted
                  // call base implementation to parse the header from payload buffer
ResponseData.PayloadPtr := SUPER^.ParseResponsePayload(ResponseData := ResponseData, Timestamp := Timestamp);

// copy parsed header to response
_response.ParSeq               := _rspHeader.ParSeq;
_response.State                := _rspHeader.State;
_response.AlarmMessageSeverity := _rspHeader.AlarmMessageSeverity;
_response.AlarmMessageCode     := _rspHeader.AlarmMessageCode;

// Check payload remaining ? 
IF ( ResponseData.IsPayloadRemaining)
THEN 
  // Get Response.RestartAccepted
 _response.RestartAccepted := ResponseData.GetBool();
  // inc parameter counter
 _parameterCnt := _parameterCnt + 1;
END_IF


// Create logging
ParseResponsePayloadLog(ResponseData := ResponseData, Timestamp := Timestamp, ParameterCnt := _parameterCnt);
                
END_METHOD

METHOD INTERNAL ParseResponsePayloadLog
VAR_INPUT
  /// Response data
  ResponseData : RobotLibraryResponseDataFB;
  /// Timestamp
  Timestamp    : SystemTime;  
  /// Parameter count
  ParameterCnt : DINT;
END_VAR
                  // Create log entry for Parameter start
CreateLogMessagePara1 ( Timestamp   := Timestamp,
                        MessageType := MessageType.CMD,
                        Severity    := Severity.DEBUG,
                        MessageCode := 0,
                        MessageText := '{1} parameter(s) to parse from the response data:',
                        Para1       := DINT_TO_STRING(ParameterCnt));
                        

// Return if no parameter is remaining...
IF ( ParameterCnt = 0 ) THEN RETURN; END_IF
// dec remaining parameter(s)                        
ParameterCnt := ParameterCnt - 1;
// Create log entry for RestartAccepted
CreateLogMessagePara1 ( Timestamp   := Timestamp,
                        MessageType := MessageType.CMD,
                        Severity    := Severity.DEBUG,
                        MessageCode := 0,
                        MessageText := 'Response.RestartAccepted = {1}',
                        Para1       :=  BOOL_TO_STRING(_response.RestartAccepted));


                
END_METHOD

METHOD PROTECTED Reset : DINT
VAR_INPUT
END_VAR
                  Reset := SUPER^.Reset();

Done               := FALSE;
Busy               := FALSE;
CommandBuffered    := FALSE;

                
END_METHOD
END_FUNCTION_BLOCK

/// Handles multiple mechanisms required for operation of the interface.
/// For maximal performance, this FB must be called after the function FB's, 
/// so that the data can be written to the fieldbus in the same cycle as the start of FB occours 
FUNCTION_BLOCK MC_RobotTaskFB EXTENDS RobotLibraryLogFB
// ------------------------------------------------------------------------- 
//  SRCI Robot Library                                                
// ------------------------------------------------------------------------- 
//                                                                           
//  Object:      RobotTaskFB                                       
//  Author:      Thorsten Brach                                                
//  Date:        2024-06-01
//
//  Description:                                              
//   
//                                                                           
//  Copyright: 
//    (C) 2024 Thorsten Brach. All rights reserved                                                                                                                                            
//             Licensed under the MIT License.
//                                                                           
//  Disclaimer:                                                                           
//    This project is provided without any guarantee and can be used for   
//    private and commercial purposes. Any use is at the user’s 
//    own risk and responsibility.
//
// -------------------------------------------------------------------------
VAR_INPUT
  /// Set TRUE (default) to initialize the interface
  Enable            : BOOL;
  /// User defined robot name
  RobotName         : STRING(20);
  /// Current System Time
  SystemTime        : SystemTime;
  /// Online Change detected
  OnlineChange      : BOOL;
  /// Axes Group ID -> is used to uniquely identify each RA on a per RC basis.
  ///
  /// For convenience, an RC with only one RA must assign ID 1 to this RA. 
  /// An RC with multiple RAs must assign numeric values 1-15 to those RAs.
  AxesGroupID       : BYTE := 0; // ToDo: Mistake in specification : ID should start with 1, but must start with 0 !  
  /// Configuration parameter
  ParCfg            : RobotTaskParCfg;
END_VAR

VAR_IN_OUT
  /// Inputs of PLC for communication from RC
  RobotInData       : ARRAY[*] OF BYTE;
  /// Outputs of PLC for communication to RC
  RobotOutData      : ARRAY[*] OF BYTE;
  ///  User data stored on the PLC according to Table 6-10
  UserData          : UserData;
  /// ToolData stored on PLC. For more information refer to 5.5.6.3
  ToolData          : ARRAY[*] OF Tool;
  /// LoadData stored on PLC.For more information refer to 5.5.6.4
  FrameData         : ARRAY[*] OF Frame;
  /// LoadData stored on PLC.For more information refer to 5.5.6.4 
  LoadData          : ARRAY[*] OF Load;
  /// Work areas stored on PLC. For more information refer to 5.5.8
  WorkAreas         : ARRAY[*] OF RobotWorkArea;
  /// Software limits stored on PLC
  SWLimits          : SWLimits;
  /// Default dynamics stored on PLC. For more information refer to 5.5.7
  DefaultDynamics   : DefaultDynamics;
  /// Reference dynamics stored on PLC. For more information refer to 5.5.7
  ReferenceDynamics : ReferenceDynamics;
  /// System log on PLC
  SystemLog         : ARRAY[0..RobotLibraryParameter.SYSTEM_LOG_MAX ] OF STRING(RobotLibraryParameter.MESSAGE_TEXT_LEN);
  /// Message buffer on the PLC - For more information refer to 5.5.11
  MessageLog        : ARRAY[0..RobotLibraryParameter.MESSAGE_LOG_MAX] OF AlarmMessage;
  /// Robot assignment of function
  AxesGroup         : AxesGroup;
END_VAR

VAR_OUTPUT
  /// FB is being processed
  Busy              : BOOL;
  /// Interface is initialized (RI state: "Initialized").
  /// For more information on RI states refer to chapter 5.5.3.1.
  Initialized       : BOOL;
  /// Server and client were successfully synchronized (RI state: "Synchronized").
  /// For more information on the synchronization mechanism refer to chapter 5.6.7.
  Synchronized      : BOOL;
  /// An error occurred
  Error             : BOOL;
  /// ErrorID reported by RC for error identification according to Table 7-1
  ErrorID           : WORD;
  ErrorIdEnum       : RobotLibraryErrorIdEnum;  
  ErrorAddTxt       : STRING(RobotLibraryConstants.MAX_ADD_TEXT_LENGTH);
  /// WarningID for warning identification reported during execution of command according to Table 7-3
  WarningID         : WORD;
  WarningIdEnum     : RobotLibraryWarningIdEnum;  
  /// InfoID for info identification reported during execution of command according to Table 7-5
  InfoID            : WORD;    
  InfoIdEnum        : RobotLibraryInfoIdEnum;    
END_VAR

VAR
  /// internal copy of configuration parameter
 _parCfg                       : RobotTaskParCfg;

  /// internal ToolData for comparation to user ToolData
 _toolData                     : ARRAY[0..RobotLibraryParameter.TOOL_MAX       -1] OF Tool;
  /// internal FrameData for comparation to user FrameData
 _frameData                    : ARRAY[0..RobotLibraryParameter.FRAME_MAX      -1] OF Frame;
  /// internal LoadData for comparation to user LoadData
 _loadData                     : ARRAY[0..RobotLibraryParameter.LOAD_MAX       -1] OF Load;
  /// internal WorkAreas for comparation to user WorkAreas
 _workAreas                    : ARRAY[0..RobotLibraryParameter.WORK_AREAS_MAX -1] OF RobotWorkArea;
  /// internal Software limits for comparation to user Software limit
 _swLimits                     : SWLimits;
  /// internal default dynamics for comparation to user default dynamics
 _defaultDynamics              : DefaultDynamics;
  /// internal reference dynamics for comparation to user reference dynamics
 _referenceDynamics            : ReferenceDynamics;

  /// FB for exchange configuration
 _exchangeConfiguration        : MC_ExchangeConfigurationFB;
  /// FB for read robot data
 _readRobotData                : MC_ReadRobotDataFB;
  /// FB for read messaged
 _readMessages                 : MC_ReadMessagesFB;  
  /// FB for read tool data
 _readToolData                 : MC_ReadToolDataFB;  
  /// FB for read frame data
 _readFrameData                : MC_ReadFrameDataFB;  
  /// FB for read load data
 _readLoadData                 : MC_ReadLoadDataFB;  
  /// FB for read work area
 _readWorkArea                 : MC_ReadWorkAreaFB;  
  /// FB for read robot software limits
 _readRobotSWLimits            : MC_ReadRobotSWLimitsFB;  
  /// FB for read robot default dynamics
 _readRobotDefaultDynamics     : MC_ReadRobotDefaultDynamicsFB;  
  /// FB for read robot reference dynamics
 _readRobotReferenceDynamics   : MC_ReadRobotReferenceDynamicsFB;  

  /// FB for write tool data
 _writeToolData                : MC_WriteToolDataFB;  
  /// FB for write frame data
 _writeFrameData               : MC_WriteFrameDataFB;  
  /// FB for write load data
 _writeLoadData                : MC_WriteLoadDataFB;  
  /// FB for write work area
 _writeWorkArea                : MC_WriteWorkAreaFB;  
  /// FB for write robot software limits
 _writeRobotSWLimits           : MC_WriteRobotSWLimitsFB;  
  /// FB for write robot default dynamics
 _writeRobotDefaultDynamics    : MC_WriteRobotDefaultDynamicsFB;  
  /// FB for write robot reference dynamics
 _writeRobotReferenceDynamics  : MC_WriteRobotReferenceDynamicsFB;  
  /// Send Buffer
  SendData                     : RobotLibrarySendDataFB;
  /// Recv Buffer
  RecvData                     : RobotLibraryRecvDataFB;
  /// Telegram 
  Telegram                     : Telegram; 
  
  /// internal step counter for command
 _stepCmd                      : DINT;
  /// internal timer for command 
  {attribute 'hide'}
 _timerCmd                     : TON;
  /// internal timeout for command
  {attribute 'hide'}
 _timeoutCmd                   : TIME := T#5S; 

  /// internal step counter for synchronisation of frame data
 _stepSyncFrameData            : DINT;
  /// internal timer for synchronisation of frame data
  {attribute 'hide'}
 _timerSyncFrameData           : TON;
  /// internal timeout for synchronisation of frame data
  {attribute 'hide'}
 _timeoutSyncFrameData         : TIME := T#5S;
   /// internal index for frame data synchronisation
 _syncIdxFrameData             : USINT;
  /// internal index for maximal amount of frames data( MIN(PLC,RC) ) 
 _syncIdxMaxFrameData          : DINT;
 
  /// internal step counter for synchronisation of load data
 _stepSyncLoadData             : DINT;
  /// internal timer for synchronisation of load data
  {attribute 'hide'}
 _timerSyncLoadData             : TON;
  /// internal timeout for synchronisation of load data
  {attribute 'hide'}
 _timeoutSyncLoadData           : TIME := T#5S; 
  /// internal index for load data synchronisation
 _syncIdxLoadData               : USINT;
  /// internal index for maximal amount of load data ( MIN(PLC,RC) ) 
 _syncIdxMaxLoadData            : DINT;

  /// internal step counter for synchronisation of tool data
 _stepSyncToolData              : DINT;
  /// internal timer for synchronisation of tool data
  {attribute 'hide'}
 _timerSyncToolData             : TON;
  /// internal timeout for synchronisation of tool data
  {attribute 'hide'}
 _timeoutSyncToolData           : TIME := T#5S; 
  /// internal index for tool data synchronisation
 _syncIdxToolData               : USINT;
  /// internal index for maximal amount of tool data ( MIN(PLC,RC) ) 
 _syncIdxMaxToolData            : DINT;

  /// internal step counter for synchronisation of work areas
 _stepSyncWorkArea            : DINT;
 /// internal timer for synchronisation of work areas
  {attribute 'hide'}
 _timerSyncWorkArea           : TON;
  /// internal timeout for synchronisation of work areas
  {attribute 'hide'}
 _timeoutSyncWorkArea         : TIME := T#5S; 
  /// internal index for WorkArea synchronisation
 _syncIdxWorkArea             : USINT;
  /// internal index for maximal amount of Work Area( MIN(PLC,RC) ) 
 _syncIdxMaxWorkArea          : DINT;
 
  /// internal step counter for synchronisation of software limits
 _stepSyncSWLimits            : DINT;
  /// internal timer for synchronisation of software limits
  {attribute 'hide'}
 _timerSyncSWLimits           : TON;
  /// internal timeout for synchronisation of software limits
  {attribute 'hide'}
 _timeoutSyncSWLimits         : TIME := T#5S; 

  /// internal step counter for synchronisation of default dynamics
 _stepSyncDefaultDynamics      : DINT;
  /// internal timer for synchronisation of default dynamics
  {attribute 'hide'}
 _timerSyncDefaultDynamics     : TON;
  /// internal timeout for synchronisation of default dynamics
  {attribute 'hide'}
 _timeoutSyncDefaultDynamics   : TIME := T#5S; 
 
  /// internal step counter for synchronisation of reference dynamics
 _stepSyncReferenceDynamics    : DINT;
  /// internal timer for synchronisation of reference dynamics
  {attribute 'hide'}
 _timerSyncReferenceDynamics   : TON;
  /// internal timeout for synchronisation of reference dynamics
  {attribute 'hide'}
 _timeoutSyncReferenceDynamics : TIME := T#5S; 


 
 
  /// Rising edge for enable
  {attribute 'hide'}
 _enable_R                    : R_TRIG;
  /// Falling edge for enable
  {attribute 'hide'}
 _enable_F                    : F_TRIG;

  /// Flag that indicated the the connection is alive (data exchange)
 _aliveBit                    : BOOL;
  /// last lifesign counter value
 _aliveValue                  : BYTE;
  /// timer for detecting alive state
 _aliveCheck                  : TON;
  /// rising edge for connection is alive
  {attribute 'hide'}
 _alive_R                     : R_TRIG;
  /// falling edge for connection is alive
  {attribute 'hide'}
 _alive_F                     : F_TRIG;
   /// last telegram state
 _lastTelegramState           : TelegramState   := TelegramState.UNDEFINED;
   /// last telegram control
 _lastTelegramControl         : ControlHalfByte := ControlHalfByte.NONE;
END_VAR

VAR // CONSTANT
  /// Lower array dimension of RobotInData
  ROBOT_IN_DATA_MIN   : DINT;
  /// Upper array dimension of RobotInData
  ROBOT_IN_DATA_MAX   : DINT;
  /// Size of RobotInData
  ROBOT_IN_DATA_SIZE  : UDINT;
  /// Lower array dimension of RobotOutData
  ROBOT_OUT_DATA_MIN  : DINT;
  /// Upper array dimension of RobotOutData
  ROBOT_OUT_DATA_MAX  : DINT;
  /// Size of RobotOutData
  ROBOT_OUT_DATA_SIZE : UDINT;
END_VAR

VAR CONSTANT
  {attribute 'hide'}
  FRAGMENT_HEADER_SIZE : UDINT := SIZEOF(TelegramPlcToRobFragmentHeader);
  /// Size of the comand header
  {attribute 'hide'}
  COMMAND_HEADER_SIZE  : UDINT := SIZEOF(TelegramPlcToRobCommandHeader);
  /// Size of the footer
  {attribute 'hide'}
  FOOTER_SIZE          : UDINT := 1;
  /// Minimal payload size for telegram
  {attribute 'hide'}
  MIN_PAYLOAD_SIZE     : UDINT := 1;
  /// Active command
  {attribute 'hide'}
  ACTIVE_CMD           : UDINT := 1;
  /// Buffered command
  {attribute 'hide'}
  BUFFER_CMD           : UDINT := 2;
  /// Empty command entry
  {attribute 'hide'}
  EMPTY_CMD_ENTRY      : AxesGroupAcyclicAcrEntryCmdBuffer := (State := BufferStateCmd.EMPTY);
  /// bitmask to mask the LifeSign out of the halfbyte
  {attribute 'hide'}
  LIFESIGN_BIT_MASK    : BYTE := 2#000_1111;   
  /// Primary sequence
  {attribute 'hide'}
  PRIMARY_SEQUENCE     : DINT := 0;
  /// Secondary sequence
  {attribute 'hide'}
  SECONDARY_SEQUENCE   : DINT := 1;  
  /// Empty Execution-Order-List entry
  {attribute 'hide'}
  EMPTY_EOL_ENTRY      : DINT := 0;
END_VAR

            // Get array dimension of RobotInData
ROBOT_IN_DATA_MIN  := LOWER_BOUND  ( RobotInData,1);
ROBOT_IN_DATA_MAX  := UPPER_BOUND  ( RobotInData,1);
ROBOT_IN_DATA_SIZE := DINT_TO_UDINT( ROBOT_IN_DATA_MAX - ROBOT_IN_DATA_MIN + 1);

// Get array dimension of RobotInData
ROBOT_OUT_DATA_MIN  := LOWER_BOUND  ( RobotOutData,1);
ROBOT_OUT_DATA_MAX  := UPPER_BOUND  ( RobotOutData,1);
ROBOT_OUT_DATA_SIZE := DINT_TO_UDINT( ROBOT_OUT_DATA_MAX - ROBOT_OUT_DATA_MIN + 1);


HandleAxesGroup              ( AxesGroup         := AxesGroup,
	                             ToolData          := ToolData, 
	                             FrameData         := FrameData, 
	                             LoadData          := LoadData, 
	                             WorkAreas         := WorkAreas, 
	                             SWLimits          := SWLimits, 
	                             DefaultDynamics   := DefaultDynamics, 
	                             ReferenceDynamics := ReferenceDynamics);
                               
HandleLifeSign               ( AxesGroup         := AxesGroup);
HandleLogMessagesAck         ( AxesGroup         := AxesGroup);
HandleInvalidFrames          ( AxesGroup         := AxesGroup, RobotInData := RobotInData);
HandleTelegramStateCtrl      (                               );
HandleAliveBit               ( RobotInData[1]                );
HandleSeqAck                 ( AxesGroup         := AxesGroup);
HandleUserData               ( AxesGroup         := AxesGroup, UserData := UserData );

HandleSync                   ( AxesGroup         := AxesGroup,
                               ToolData          := ToolData,
                               FrameData         := FrameData,
                               LoadData          := LoadData,
                               WorkAreas         := WorkAreas,
                               SWLimits          := SWLimits,
                               DefaultDynamics   := DefaultDynamics,
                               ReferenceDynamics := ReferenceDynamics);

OnCall                       ( AxesGroup         := AxesGroup);
OnExecRun                    ( AxesGroup         := AxesGroup);

AxesGroupToTelegram          ( AxesGroup         := AxesGroup );

CreateSendPayload            ( AxesGroup         := AxesGroup, RobotOutData := RobotOutData );
ParseRecvPayload             ( AxesGroup         := AxesGroup, RobotInData  := RobotInData); 

AxesGroupFromTelegram        ( AxesGroup         := AxesGroup);


// call internal functionblocks
_exchangeConfiguration      ( Name := RobotName, ExecMode := ExecutionMode.PARALLEL, Priority := PriorityLevel.NORMAL, AxesGroup := AxesGroup );
_readRobotData              ( Name := RobotName, ExecMode := ExecutionMode.PARALLEL, Priority := PriorityLevel.NORMAL, AxesGroup := AxesGroup );
_readMessages               ( Name := RobotName, ExecMode := ExecutionMode.PARALLEL, Priority := PriorityLevel.NORMAL, AxesGroup := AxesGroup );
_readToolData               ( Name := RobotName, ExecMode := ExecutionMode.PARALLEL, Priority := PriorityLevel.NORMAL, AxesGroup := AxesGroup );
_readFrameData              ( Name := RobotName, ExecMode := ExecutionMode.PARALLEL, Priority := PriorityLevel.NORMAL, AxesGroup := AxesGroup );
_readLoadData               ( Name := RobotName, ExecMode := ExecutionMode.PARALLEL, Priority := PriorityLevel.NORMAL, AxesGroup := AxesGroup );
_readWorkArea               ( Name := RobotName, ExecMode := ExecutionMode.PARALLEL, Priority := PriorityLevel.NORMAL, AxesGroup := AxesGroup );  
_readRobotSWLimits          ( Name := RobotName, ExecMode := ExecutionMode.PARALLEL, Priority := PriorityLevel.NORMAL, AxesGroup := AxesGroup );  
_readRobotDefaultDynamics   ( Name := RobotName, ExecMode := ExecutionMode.PARALLEL, Priority := PriorityLevel.NORMAL, AxesGroup := AxesGroup );
_readRobotReferenceDynamics ( Name := RobotName, ExecMode := ExecutionMode.PARALLEL, Priority := PriorityLevel.NORMAL, AxesGroup := AxesGroup );
_writeToolData              ( Name := RobotName, ExecMode := ExecutionMode.PARALLEL, Priority := PriorityLevel.NORMAL, AxesGroup := AxesGroup );  
_writeFrameData             ( Name := RobotName, ExecMode := ExecutionMode.PARALLEL, Priority := PriorityLevel.NORMAL, AxesGroup := AxesGroup );  
_writeLoadData              ( Name := RobotName, ExecMode := ExecutionMode.PARALLEL, Priority := PriorityLevel.NORMAL, AxesGroup := AxesGroup );  
_writeWorkArea              ( Name := RobotName, ExecMode := ExecutionMode.PARALLEL, Priority := PriorityLevel.NORMAL, AxesGroup := AxesGroup );  
_writeRobotSWLimits         ( Name := RobotName, ExecMode := ExecutionMode.PARALLEL, Priority := PriorityLevel.NORMAL, AxesGroup := AxesGroup );  
_writeRobotDefaultDynamics  ( Name := RobotName, ExecMode := ExecutionMode.PARALLEL, Priority := PriorityLevel.NORMAL, AxesGroup := AxesGroup );  
_writeRobotReferenceDynamics( Name := RobotName, ExecMode := ExecutionMode.PARALLEL, Priority := PriorityLevel.NORMAL, AxesGroup := AxesGroup );  


// Update SystemLog and MessageLog
SystemLog  := AxesGroup.MessageLog.SystemLogs;
MessageLog := AxesGroup.MessageLog.Messages;
          

METHOD PRIVATE AxesGroupFromTelegram
VAR_IN_OUT
  /// Robot assignment of function
  AxesGroup    : AxesGroup;
END_VAR
                  AxesGroupFromTelegramCyclic         (AxesGroup := AxesGroup);
AxesGroupFromTelegramCyclicOptional (AxesGroup := AxesGroup);
                
END_METHOD

METHOD PRIVATE AxesGroupFromTelegramCyclic
VAR_IN_OUT
  /// Robot assignment of function
  AxesGroup : AxesGroup;
END_VAR
                  // ---------------------------------
// Mapp Telegramm to AxesGroup Data  
// ---------------------------------
AxesGroup.Cyclic.RobToPlc.SRCIVersion    := Telegram.RobToPlc.Header.SRCIVersion ;
AxesGroup.Cyclic.RobToPlc.LifeSign       := Telegram.RobToPlc.Header.LifeSign ;
AxesGroup.Cyclic.RobToPlc.TelegramState  := Telegram.RobToPlc.Header.TelegramState ;
AxesGroup.Cyclic.RobToPlc.StatusRobotArm := DwordToRaStatusWord(Telegram.RobToPlc.Header.StatusRobotArm);
AxesGroup.Cyclic.RobToPlc.Override       := Telegram.RobToPlc.Header.Override ;
                
END_METHOD

METHOD PRIVATE AxesGroupFromTelegramCyclicOptional
VAR_IN_OUT
  /// Robot assignment of function
  AxesGroup: AxesGroup;
END_VAR
                  // Sub ProgramData {{{
AxesGroup.CyclicOptional.RobToPlc.SubProgramData.Data := Telegram.RobToPlc.CyclicOptional.SubProgramData.Data;
// }}}


// Cartesian position {{{
AxesGroup.CyclicOptional.RobToPlc.CartesianPosition.Active                   :=                                     AxesGroup.CyclicOptional.RobToPlc.CartesianPosition.Active;
AxesGroup.CyclicOptional.RobToPlc.CartesianPosition.X                        :=                                      Telegram.RobToPlc.CyclicOptional.CartesianPosition.X;
AxesGroup.CyclicOptional.RobToPlc.CartesianPosition.Y                        :=                                      Telegram.RobToPlc.CyclicOptional.CartesianPosition.Y;
AxesGroup.CyclicOptional.RobToPlc.CartesianPosition.Z                        :=                                      Telegram.RobToPlc.CyclicOptional.CartesianPosition.Z;
AxesGroup.CyclicOptional.RobToPlc.CartesianPosition.Rx                       :=                                      Telegram.RobToPlc.CyclicOptional.CartesianPosition.Rx;
AxesGroup.CyclicOptional.RobToPlc.CartesianPosition.Ry                       :=                                      Telegram.RobToPlc.CyclicOptional.CartesianPosition.Ry;
AxesGroup.CyclicOptional.RobToPlc.CartesianPosition.Rz                       :=                                      Telegram.RobToPlc.CyclicOptional.CartesianPosition.Rz;
AxesGroup.CyclicOptional.RobToPlc.CartesianPosition.Config.Shoulder          :=              WordToArmConfigShoulder(Telegram.RobToPlc.CyclicOptional.CartesianPosition.Config);
AxesGroup.CyclicOptional.RobToPlc.CartesianPosition.Config.Elbow             :=              WordToArmConfigElbow   (Telegram.RobToPlc.CyclicOptional.CartesianPosition.Config);
AxesGroup.CyclicOptional.RobToPlc.CartesianPosition.Config.Wrist             :=              WordToArmConfigWrist   (Telegram.RobToPlc.CyclicOptional.CartesianPosition.Config);
AxesGroup.CyclicOptional.RobToPlc.CartesianPosition.TurnNumber.J1Turns       := BYTE_TO_SINT(GetHalfeByteLo         (Telegram.RobToPlc.CyclicOptional.CartesianPosition.Turns_J2_J1));
AxesGroup.CyclicOptional.RobToPlc.CartesianPosition.TurnNumber.J2Turns       := BYTE_TO_SINT(GetHalfeByteHi         (Telegram.RobToPlc.CyclicOptional.CartesianPosition.Turns_J2_J1));
AxesGroup.CyclicOptional.RobToPlc.CartesianPosition.TurnNumber.J3Turns       := BYTE_TO_SINT(GetHalfeByteLo         (Telegram.RobToPlc.CyclicOptional.CartesianPosition.Turns_J4_J3));
AxesGroup.CyclicOptional.RobToPlc.CartesianPosition.TurnNumber.J4Turns       := BYTE_TO_SINT(GetHalfeByteHi         (Telegram.RobToPlc.CyclicOptional.CartesianPosition.Turns_J4_J3));
AxesGroup.CyclicOptional.RobToPlc.CartesianPosition.TurnNumber.J5Turns       := BYTE_TO_SINT(GetHalfeByteLo         (Telegram.RobToPlc.CyclicOptional.CartesianPosition.Turns_J6_J5));
AxesGroup.CyclicOptional.RobToPlc.CartesianPosition.TurnNumber.J6Turns       := BYTE_TO_SINT(GetHalfeByteHi         (Telegram.RobToPlc.CyclicOptional.CartesianPosition.Turns_J6_J5));
AxesGroup.CyclicOptional.RobToPlc.CartesianPosition.TurnNumber.E1Turns       := BYTE_TO_SINT                        (Telegram.RobToPlc.CyclicOptional.CartesianPosition.Turns_E1);
AxesGroup.CyclicOptional.RobToPlc.CartesianPosition.E1                       :=                                      Telegram.RobToPlc.CyclicOptional.CartesianPosition.E1;
AxesGroup.CyclicOptional.RobToPlc.CartesianPosition.CoordinateSystem.ToolNo  :=                                      Telegram.RobToPlc.CyclicOptional.CartesianPosition.CurrentlyUsedToolNo;
AxesGroup.CyclicOptional.RobToPlc.CartesianPosition.CoordinateSystem.FrameNo :=                                      Telegram.RobToPlc.CyclicOptional.CartesianPosition.CurrentlyUsedFrameNo;
// }}}


// Joint position {{{
AxesGroup.CyclicOptional.RobToPlc.JointPosition.Active := AxesGroup.CyclicOptional.RobToPlc.JointPosition.Active;
AxesGroup.CyclicOptional.RobToPlc.JointPosition.J1     :=  Telegram.RobToPlc.CyclicOptional.JointPosition.J1;
AxesGroup.CyclicOptional.RobToPlc.JointPosition.J2     :=  Telegram.RobToPlc.CyclicOptional.JointPosition.J2;
AxesGroup.CyclicOptional.RobToPlc.JointPosition.J3     :=  Telegram.RobToPlc.CyclicOptional.JointPosition.J3;
AxesGroup.CyclicOptional.RobToPlc.JointPosition.J4     :=  Telegram.RobToPlc.CyclicOptional.JointPosition.J4;
AxesGroup.CyclicOptional.RobToPlc.JointPosition.J5     :=  Telegram.RobToPlc.CyclicOptional.JointPosition.J5;
AxesGroup.CyclicOptional.RobToPlc.JointPosition.J6     :=  Telegram.RobToPlc.CyclicOptional.JointPosition.J6;
AxesGroup.CyclicOptional.RobToPlc.JointPosition.E1     :=  Telegram.RobToPlc.CyclicOptional.JointPosition.E1;
// }}}

// Force {{{
AxesGroup.CyclicOptional.RobToPlc.Force.Active          := AxesGroup.CyclicOptional.RobToPlc.Force.Active;
AxesGroup.CyclicOptional.RobToPlc.Force.X               :=  Telegram.RobToPlc.CyclicOptional.Force.X;
AxesGroup.CyclicOptional.RobToPlc.Force.Y               :=  Telegram.RobToPlc.CyclicOptional.Force.Y;
AxesGroup.CyclicOptional.RobToPlc.Force.Z               :=  Telegram.RobToPlc.CyclicOptional.Force.Z;
AxesGroup.CyclicOptional.RobToPlc.Force.Rx              :=  Telegram.RobToPlc.CyclicOptional.Force.Rx;
AxesGroup.CyclicOptional.RobToPlc.Force.Ry              :=  Telegram.RobToPlc.CyclicOptional.Force.Ry;
AxesGroup.CyclicOptional.RobToPlc.Force.Rz              :=  Telegram.RobToPlc.CyclicOptional.Force.Rz;
// }}}

// Current {{{
AxesGroup.CyclicOptional.RobToPlc.Current.Active        := AxesGroup.CyclicOptional.RobToPlc.Current.Active;
AxesGroup.CyclicOptional.RobToPlc.Current.J1            :=  Telegram.RobToPlc.CyclicOptional.Current.J1;
AxesGroup.CyclicOptional.RobToPlc.Current.J2            :=  Telegram.RobToPlc.CyclicOptional.Current.J2;
AxesGroup.CyclicOptional.RobToPlc.Current.J3            :=  Telegram.RobToPlc.CyclicOptional.Current.J3;
AxesGroup.CyclicOptional.RobToPlc.Current.J4            :=  Telegram.RobToPlc.CyclicOptional.Current.J4;
AxesGroup.CyclicOptional.RobToPlc.Current.J5            :=  Telegram.RobToPlc.CyclicOptional.Current.J5;
AxesGroup.CyclicOptional.RobToPlc.Current.J6            :=  Telegram.RobToPlc.CyclicOptional.Current.J6;
// }}}


// Two Sequences {{{
// }}}

// Cartesian Position Extended
AxesGroup.CyclicOptional.RobToPlc.CartesianPositionExt.Active := AxesGroup.CyclicOptional.RobToPlc.CartesianPositionExt.Active;
AxesGroup.CyclicOptional.RobToPlc.CartesianPositionExt.E2     :=  Telegram.RobToPlc.CyclicOptional.CartesianPositionExt.E2;
AxesGroup.CyclicOptional.RobToPlc.CartesianPositionExt.E3     :=  Telegram.RobToPlc.CyclicOptional.CartesianPositionExt.E3;
AxesGroup.CyclicOptional.RobToPlc.CartesianPositionExt.E4     :=  Telegram.RobToPlc.CyclicOptional.CartesianPositionExt.E4;
AxesGroup.CyclicOptional.RobToPlc.CartesianPositionExt.E5     :=  Telegram.RobToPlc.CyclicOptional.CartesianPositionExt.E5;
AxesGroup.CyclicOptional.RobToPlc.CartesianPositionExt.E6     :=  Telegram.RobToPlc.CyclicOptional.CartesianPositionExt.E6;

// Joint Position Extended
AxesGroup.CyclicOptional.RobToPlc.JointPositionExt.Active     := AxesGroup.CyclicOptional.RobToPlc.JointPositionExt.Active;
AxesGroup.CyclicOptional.RobToPlc.JointPositionExt.E2         :=  Telegram.RobToPlc.CyclicOptional.JointPositionExt.E2;
AxesGroup.CyclicOptional.RobToPlc.JointPositionExt.E3         :=  Telegram.RobToPlc.CyclicOptional.JointPositionExt.E3;
AxesGroup.CyclicOptional.RobToPlc.JointPositionExt.E4         :=  Telegram.RobToPlc.CyclicOptional.JointPositionExt.E4;
AxesGroup.CyclicOptional.RobToPlc.JointPositionExt.E5         :=  Telegram.RobToPlc.CyclicOptional.JointPositionExt.E5;
AxesGroup.CyclicOptional.RobToPlc.JointPositionExt.E6         :=  Telegram.RobToPlc.CyclicOptional.JointPositionExt.E6;

// Force Extended
AxesGroup.CyclicOptional.RobToPlc.ForceExt.Active             := AxesGroup.CyclicOptional.RobToPlc.ForceExt.Active;
AxesGroup.CyclicOptional.RobToPlc.ForceExt.E1                 :=  Telegram.RobToPlc.CyclicOptional.ForceExt.E1;
AxesGroup.CyclicOptional.RobToPlc.ForceExt.E2                 :=  Telegram.RobToPlc.CyclicOptional.ForceExt.E2;
AxesGroup.CyclicOptional.RobToPlc.ForceExt.E3                 :=  Telegram.RobToPlc.CyclicOptional.ForceExt.E3;
AxesGroup.CyclicOptional.RobToPlc.ForceExt.E4                 :=  Telegram.RobToPlc.CyclicOptional.ForceExt.E4;
AxesGroup.CyclicOptional.RobToPlc.ForceExt.E5                 :=  Telegram.RobToPlc.CyclicOptional.ForceExt.E5;
AxesGroup.CyclicOptional.RobToPlc.ForceExt.E6                 :=  Telegram.RobToPlc.CyclicOptional.ForceExt.E6;

// Current Extended
AxesGroup.CyclicOptional.RobToPlc.CurrentExt.Active           := AxesGroup.CyclicOptional.RobToPlc.CurrentExt.Active;
AxesGroup.CyclicOptional.RobToPlc.CurrentExt.E1               :=  Telegram.RobToPlc.CyclicOptional.CurrentExt.E1;
AxesGroup.CyclicOptional.RobToPlc.CurrentExt.E2               :=  Telegram.RobToPlc.CyclicOptional.CurrentExt.E2;
AxesGroup.CyclicOptional.RobToPlc.CurrentExt.E3               :=  Telegram.RobToPlc.CyclicOptional.CurrentExt.E3;
AxesGroup.CyclicOptional.RobToPlc.CurrentExt.E4               :=  Telegram.RobToPlc.CyclicOptional.CurrentExt.E4;
AxesGroup.CyclicOptional.RobToPlc.CurrentExt.E5               :=  Telegram.RobToPlc.CyclicOptional.CurrentExt.E5;
AxesGroup.CyclicOptional.RobToPlc.CurrentExt.E6               :=  Telegram.RobToPlc.CyclicOptional.CurrentExt.E6;
                
END_METHOD

METHOD PRIVATE AxesGroupToTelegram : DINT
VAR_IN_OUT
  /// Robot assignment of function
  AxesGroup : AxesGroup;
END_VAR

VAR 
  /// internal index
 _idx                       : DINT;
  /// internal sequence index
 _seqIdx                    : DINT;
  /// internal fragment index
 _fragIdx                   : DINT;
  /// internal register index
 _regIdx                    : DINT;
  /// internal execution order list index
 _listIdx                   : DINT := 1;
  /// internal payload pointer
 _payLoadPtr                : DWORD;
  /// internal fragment action
 _fragmentAction            : FragmentAction;
  /// internal fragment action as string
 _fragmentActionString      : STRING;
  /// maximount amount of bytes per sequence
  SEQUENCE_MAX_PAYLOAD_SIZE : UDINT;
END_VAR
                  IF ( AxesGroup.State.NewSEQ[0]) {warning 'Handle 2nd sequence'}
THEN
  // delete old telegram data 
  SysDepMemSet(pDest := ADR(Telegram.PlcToRob), Value := 0 , DataLen := SIZEOF(Telegram.PlcToRob));
END_IF
  
AxesGroupToTelegramHeader        (AxesGroup := AxesGroup);
AxesGroupToTelegramCyclic        (AxesGroup := AxesGroup);
AxesGroupToTelegramCyclicOptional(AxesGroup := AxesGroup);
AxesGroupToTelegramSequence      (AxesGroup := AxesGroup);
AxesGroupToTelegramFooter        (AxesGroup := AxesGroup);
AxesGroupToTelegramLogging       (AxesGroup := AxesGroup);
                
END_METHOD

METHOD PRIVATE AxesGroupToTelegramCyclic : DINT
VAR_IN_OUT
  /// Robot assignment of function
  AxesGroup : AxesGroup;
END_VAR
                  IF (AxesGroup.Cyclic.PlcToRob.ToolNo = -1 )
THEN
  Telegram.PlcToRob.Cyclic.ToolNo  := 16#FF;
ELSE
  Telegram.PlcToRob.Cyclic.ToolNo  := INT_TO_BYTE(AxesGroup.Cyclic.PlcToRob.ToolNo); 
END_IF

IF (AxesGroup.Cyclic.PlcToRob.FrameNo = -1 )
THEN
  Telegram.PlcToRob.Cyclic.FrameNo  := 16#FF;
ELSE
  Telegram.PlcToRob.Cyclic.FrameNo  := INT_TO_BYTE(AxesGroup.Cyclic.PlcToRob.FrameNo); 
END_IF
                
END_METHOD

METHOD PRIVATE AxesGroupToTelegramCyclicOptional : DINT
VAR_IN_OUT
  /// Robot assignment of function
  AxesGroup : AxesGroup;
END_VAR
                  // AxesGroup.CyclicOptional.PlcToRob.SubProgramData {{{
IF (AxesGroup.CyclicOptional.PlcToRob.SubProgramData.Active)
THEN
  Telegram.PlcToRob.CyclicOptional.SubProgramData.Data := AxesGroup.CyclicOptional.PlcToRob.SubProgramData.Data; 
END_IF
// }}}

// AxesGroup.CyclicOptional.PlcToRob.CartesianPosition  {{{  
IF (AxesGroup.CyclicOptional.PlcToRob.CartesianPosition.Active)
THEN
  Telegram.PlcToRob.CyclicOptional.CartesianPosition.X           :=                  AxesGroup.CyclicOptional.PlcToRob.CartesianPosition.X;  
  Telegram.PlcToRob.CyclicOptional.CartesianPosition.Y           :=                  AxesGroup.CyclicOptional.PlcToRob.CartesianPosition.Y;  
  Telegram.PlcToRob.CyclicOptional.CartesianPosition.Z           :=                  AxesGroup.CyclicOptional.PlcToRob.CartesianPosition.Z;
  Telegram.PlcToRob.CyclicOptional.CartesianPosition.Rx          :=                  AxesGroup.CyclicOptional.PlcToRob.CartesianPosition.Rx;  
  Telegram.PlcToRob.CyclicOptional.CartesianPosition.Ry          :=                  AxesGroup.CyclicOptional.PlcToRob.CartesianPosition.Ry;  
  Telegram.PlcToRob.CyclicOptional.CartesianPosition.Rz          :=                  AxesGroup.CyclicOptional.PlcToRob.CartesianPosition.Rz;
  Telegram.PlcToRob.CyclicOptional.CartesianPosition.Turns_J2_J1 := CombineHalfSints(AxesGroup.CyclicOptional.PlcToRob.CartesianPosition.TurnNumber.J2Turns, 
                                                                                     AxesGroup.CyclicOptional.PlcToRob.CartesianPosition.TurnNumber.J1Turns);
  Telegram.PlcToRob.CyclicOptional.CartesianPosition.Turns_J4_J3 := CombineHalfSints(AxesGroup.CyclicOptional.PlcToRob.CartesianPosition.TurnNumber.J4Turns, 
                                                                                     AxesGroup.CyclicOptional.PlcToRob.CartesianPosition.TurnNumber.J3Turns);
  Telegram.PlcToRob.CyclicOptional.CartesianPosition.Turns_J6_J5 := CombineHalfSints(AxesGroup.CyclicOptional.PlcToRob.CartesianPosition.TurnNumber.J6Turns, 
                                                                                     AxesGroup.CyclicOptional.PlcToRob.CartesianPosition.TurnNumber.J5Turns);
  Telegram.PlcToRob.CyclicOptional.CartesianPosition.Turns_E1    := SINT_TO_BYTE    (AxesGroup.CyclicOptional.PlcToRob.CartesianPosition.TurnNumber.E1Turns);
END_IF  
// }}}
  
// AxesGroup.CyclicOptional.PlcToRob.CartesianPositionExt {{{ 
IF ( AxesGroup.CyclicOptional.PlcToRob.CartesianPositionExt.Active) 
THEN
  Telegram.PlcToRob.CyclicOptional.CartesianPositionExt.E2 := AxesGroup.CyclicOptional.PlcToRob.CartesianPositionExt.E2;  
  Telegram.PlcToRob.CyclicOptional.CartesianPositionExt.E3 := AxesGroup.CyclicOptional.PlcToRob.CartesianPositionExt.E3;  
  Telegram.PlcToRob.CyclicOptional.CartesianPositionExt.E4 := AxesGroup.CyclicOptional.PlcToRob.CartesianPositionExt.E4;  
  Telegram.PlcToRob.CyclicOptional.CartesianPositionExt.E5 := AxesGroup.CyclicOptional.PlcToRob.CartesianPositionExt.E5;  
  Telegram.PlcToRob.CyclicOptional.CartesianPositionExt.E6 := AxesGroup.CyclicOptional.PlcToRob.CartesianPositionExt.E6;  
END_IF
// }}}

// AxesGroup.CyclicOptional.PlcToRob.JointPosition {{{
IF ( AxesGroup.CyclicOptional.PlcToRob.JointPosition.Active) 
THEN
  Telegram.PlcToRob.CyclicOptional.JointPosition.J1 := AxesGroup.CyclicOptional.PlcToRob.JointPosition.J1;
  Telegram.PlcToRob.CyclicOptional.JointPosition.J2 := AxesGroup.CyclicOptional.PlcToRob.JointPosition.J2;
  Telegram.PlcToRob.CyclicOptional.JointPosition.J3 := AxesGroup.CyclicOptional.PlcToRob.JointPosition.J3;
  Telegram.PlcToRob.CyclicOptional.JointPosition.J4 := AxesGroup.CyclicOptional.PlcToRob.JointPosition.J4;
  Telegram.PlcToRob.CyclicOptional.JointPosition.J5 := AxesGroup.CyclicOptional.PlcToRob.JointPosition.J5;
  Telegram.PlcToRob.CyclicOptional.JointPosition.J6 := AxesGroup.CyclicOptional.PlcToRob.JointPosition.J6;
  Telegram.PlcToRob.CyclicOptional.JointPosition.E1 := AxesGroup.CyclicOptional.PlcToRob.JointPosition.E1;
END_IF
// }}}

// AxesGroup.CyclicOptional.PlcToRob.JointPositionExt {{{
IF ( AxesGroup.CyclicOptional.PlcToRob.JointPositionExt.Active) 
THEN
  Telegram.PlcToRob.CyclicOptional.JointPositionExt.E2 := AxesGroup.CyclicOptional.PlcToRob.JointPositionExt.E2;
  Telegram.PlcToRob.CyclicOptional.JointPositionExt.E3 := AxesGroup.CyclicOptional.PlcToRob.JointPositionExt.E3;  
  Telegram.PlcToRob.CyclicOptional.JointPositionExt.E4 := AxesGroup.CyclicOptional.PlcToRob.JointPositionExt.E4;
  Telegram.PlcToRob.CyclicOptional.JointPositionExt.E5 := AxesGroup.CyclicOptional.PlcToRob.JointPositionExt.E5;
  Telegram.PlcToRob.CyclicOptional.JointPositionExt.E6 := AxesGroup.CyclicOptional.PlcToRob.JointPositionExt.E6;        
END_IF  
// }}}
     
// AxesGroup.CyclicOptional.PlcToRob.Force {{{
IF ( AxesGroup.CyclicOptional.PlcToRob.Force.Active) 
THEN
  Telegram.PlcToRob.CyclicOptional.Force.X  := AxesGroup.CyclicOptional.PlcToRob.Force.X;
  Telegram.PlcToRob.CyclicOptional.Force.Y  := AxesGroup.CyclicOptional.PlcToRob.Force.Y;
  Telegram.PlcToRob.CyclicOptional.Force.Z  := AxesGroup.CyclicOptional.PlcToRob.Force.Z;
  Telegram.PlcToRob.CyclicOptional.Force.Rx := AxesGroup.CyclicOptional.PlcToRob.Force.Rx;
  Telegram.PlcToRob.CyclicOptional.Force.Ry := AxesGroup.CyclicOptional.PlcToRob.Force.Ry;
  Telegram.PlcToRob.CyclicOptional.Force.Rz := AxesGroup.CyclicOptional.PlcToRob.Force.Rz;
END_IF  
// }}}
                    
// AxesGroup.CyclicOptional.PlcToRob.ForceExt {{{
IF ( AxesGroup.CyclicOptional.PlcToRob.ForceExt.Active) 
THEN
  Telegram.PlcToRob.CyclicOptional.ForceExt.E1 := AxesGroup.CyclicOptional.PlcToRob.ForceExt.E1;
  Telegram.PlcToRob.CyclicOptional.ForceExt.E2 := AxesGroup.CyclicOptional.PlcToRob.ForceExt.E2;
  Telegram.PlcToRob.CyclicOptional.ForceExt.E3 := AxesGroup.CyclicOptional.PlcToRob.ForceExt.E3;
  Telegram.PlcToRob.CyclicOptional.ForceExt.E4 := AxesGroup.CyclicOptional.PlcToRob.ForceExt.E4;
  Telegram.PlcToRob.CyclicOptional.ForceExt.E5 := AxesGroup.CyclicOptional.PlcToRob.ForceExt.E5;
  Telegram.PlcToRob.CyclicOptional.ForceExt.E6 := AxesGroup.CyclicOptional.PlcToRob.ForceExt.E6;
END_IF                    
// }}}
                
END_METHOD

METHOD PRIVATE AxesGroupToTelegramFooter : DINT
VAR_IN_OUT
  /// Robot assignment of function
  AxesGroup : AxesGroup;
END_VAR
                  Telegram.PlcToRob.Footer.LifeSign := GetHalfeByteLo(Telegram.PlcToRob.Header.FastStop_LifeSign);  
                
END_METHOD

METHOD PRIVATE AxesGroupToTelegramHeader : DINT
VAR_IN_OUT
  /// Robot assignment of function
  AxesGroup : AxesGroup;
END_VAR
                  Telegram.PlcToRob.Header.SRCIVersion               := VersionToByte(AxesGroup.Cyclic.PlcToRob.SRCIVersion);
Telegram.PlcToRob.Header.FastStop_LifeSign         := CombineHalfBytes( HalfByteHi := AxesGroup.Cyclic.PlcToRob.FastStop, HalfByteLo := AxesGroup.Cyclic.PlcToRob.LifeSign );
Telegram.PlcToRob.Header.TelegramLengthPlcToRob    := ParCfg.Com.TelegramLengthPlcToRob;
Telegram.PlcToRob.Header.TelegramLengthRobToPlc    := ParCfg.Com.TelegramLengthRobToPlc;
Telegram.PlcToRob.Header.AxesGroupID_Control       := CombineHalfBytes(HalfByteHi := AxesGroup.Cyclic.PlcToRob.AxesGroupID, HalfByteLo := AxesGroup.Cyclic.PlcToRob.Control);
Telegram.PlcToRob.Header.Reserved                  := 0;
Telegram.PlcToRob.Header.TelegramNumberPlcToRob    := PlcOptionalCyclicToUint(AxesGroup.Parameter.Plc.OptionalCyclic);
Telegram.PlcToRob.Header.TelegramNumberRobToPlc    := RobOptionalCyclicToUint(AxesGroup.Parameter.Rob.OptionalCyclic);
Telegram.PlcToRob.Header.ClientDate                := AxesGroup.Cyclic.PlcToRob.ClientDate;
Telegram.PlcToRob.Header.ClientTime                := AxesGroup.Cyclic.PlcToRob.ClientTime;
                
END_METHOD

METHOD PRIVATE AxesGroupToTelegramLogging : DINT
VAR_IN_OUT
  /// Robot assignment of function
  AxesGroup : AxesGroup;
END_VAR

VAR 
  /// internal sequence index
 _seqIdx                    : DINT;
  /// internal fragment index
 _fragIdx                   : DINT;
END_VAR
                  FOR _seqIdx := 0 TO AxesGroup.State.SequenceCountSend
DO
  // check new data ? 
  IF ( AxesGroup.State.NewSEQ[_seqIdx] )
  THEN
    IF ( Telegram.PlcToRob.Sequence[_seqIdx].Header.PayloadLength > 0 ) 
    THEN
      // Create log entry
      CreateLogMessagePara4 ( Timestamp   := SystemTime,
                              MessageType := MessageType.CMD,
                              Severity    := Severity.DEBUG,
                              MessageCode := 0,
                              MessageText := 'SendData: SEQ = {1}, added Sequence [{2}] with PayloadLength = {3}, HeaderLength = {4}',
                              Para1       :=  UINT_TO_STRING(Telegram.PlcToRob.Sequence[_seqIdx].Header.SEQ_ACK),
                              Para2       :=  DINT_TO_STRING(_seqIdx),
                              Para3       :=  UINT_TO_STRING(Telegram.PlcToRob.Sequence[_seqIdx].Header.PayloadLength),
                              Para4       :=  DINT_TO_STRING(SIZEOF(Telegram.PlcToRob.Sequence[_seqIdx].Header)));
    END_IF
    
    FOR _fragIdx := 0 TO AxesGroup.State.FragmentCountSend[_seqIdx]
    DO
      IF ( Telegram.PlcToRob.Sequence[_seqIdx].Fragment[_fragIdx].Header.PayloadLength > 0 )
      THEN
        // Create log entry
        CreateLogMessagePara6 ( Timestamp   := SystemTime,
                                MessageType := MessageType.CMD,
                                Severity    := Severity.DEBUG,
                                MessageCode := 0,
                                MessageText := 'SendData: added Fragment [{1}] with PayloadLength = {2}, HeaderLength = {3}, CmdID <{4}>, Cmd <{5}> Fragment-Action Bits:{6}' ,
                                Para1       := DINT_TO_STRING(_fragIdx),
                                Para2       := UINT_TO_STRING            (Telegram.PlcToRob.Sequence[_seqIdx].Fragment[_fragIdx].Header.PayloadLength),
                                Para3       := DINT_TO_STRING(SIZEOF     (Telegram.PlcToRob.Sequence[_seqIdx].Fragment[_fragIdx].Header)),                                
                                Para4       := UINT_TO_STRING            (Telegram.PlcToRob.Sequence[_seqIdx].Fragment[_fragIdx].Header.CmdID),
                                Para5       := CMD_TYPE_TO_STRING        (Telegram.PlcToRob.Sequence[_seqIdx].Fragment[_fragIdx].Command.Header.CmdType),
                                Para6       := FRAGMENT_ACTION_TO_STRING (Telegram.PlcToRob.Sequence[_seqIdx].Fragment[_fragIdx].Header.FragmentAction)); 

        // Create log entry
        CreateLogMessagePara2 ( Timestamp   := SystemTime,
                                MessageType := MessageType.CMD,
                                Severity    := Severity.DEBUG,
                                MessageCode := 0,
                                MessageText := 'SendData: added Fragment [{1}] will be executed with ExecMode = [{2}]' ,
                                Para1       := DINT_TO_STRING(_fragIdx),
                                Para2       := EXECUTION_MODE_TO_STRING(Telegram.PlcToRob.Sequence[_seqIdx].Fragment[_fragIdx].Command.Header.ExecMode));

      END_IF
    END_FOR
  END_IF
END_FOR
                
END_METHOD

METHOD PRIVATE AxesGroupToTelegramSequence : DINT
VAR_IN_OUT
  /// Robot assignment of function
  AxesGroup : AxesGroup;
END_VAR

VAR 
  /// internal index
 _idx                       : DINT;
  /// internal sequence index
 _seqIdx                    : DINT;
   /// Amount of sequences
 _seqCount                  : DINT;

  /// internal fragment index
 _fragIdx                   : DINT;
  /// internal register index
 _regIdx                    : DINT;
  /// internal execution order list index
 _listIdx                   : DINT := 1;
  /// internal payload pointer
 _payLoadPtr                : DWORD;
  /// internal fragment action
 _fragmentAction            : FragmentAction;
  /// internal fragment action as string
 _fragmentActionString      : STRING;
  /// maximount amount of bytes per sequence
  SEQUENCE_MAX_PAYLOAD_SIZE : UDINT;
  
  /// current length of telegram 
 _telegramLengthCurrent    : UINT;
END_VAR
                  // Check 2nd sequence active ? 
IF ( _parCfg.Com.TwoSequences )
THEN
  // inc sequence counter
 _seqCount := _seqCount + 1;
  
  SEQUENCE_MAX_PAYLOAD_SIZE := CalculateSequencePayloadMax(AxesGroup := AxesGroup, 
                                                           Direction := ComDirection.PLC_TO_ROB, 
                                                           Sequence  := SequenceFlag.SECONDARY_SEQUENCE ) - FOOTER_SIZE;
ELSE
  SEQUENCE_MAX_PAYLOAD_SIZE := CalculateSequencePayloadMax(AxesGroup := AxesGroup, 
                                                           Direction := ComDirection.PLC_TO_ROB, 
                                                           Sequence  := SequenceFlag.PRIMARY_SEQUENCE   ) - FOOTER_SIZE;
END_IF   


FOR _seqIdx := 0 TO _seqCount
DO
  // set current SEQ / ACk index
  Telegram.PlcToRob.Sequence[_seqIdx].Header.SEQ_ACK := AxesGroup.State.CurrentSEQ[_seqIdx];

  // only update telegram content if a new sequence SEQ is set
  IF ( AxesGroup.State.NewSEQ[_seqIdx] ) 
  THEN
    // only reset counters in case of new telegram to send  
    AxesGroup.State.SequenceCountSend := 0;
    AxesGroup.State.FragmentCountSend[_seqIdx] := 0;
    
    // calc current telegram payload length
   _telegramLengthCurrent := CalculateTelegramLengthPlcToRob(AxesGroup := AxesGroup);
    
    // Bedingung anpassen und TWO_SEQUENCES berücksichtigen
    WHILE (( _parCfg.Com.TelegramLengthPlcToRob - _telegramLengthCurrent ) >= FRAGMENT_HEADER_SIZE + MIN_PAYLOAD_SIZE ) 
    DO
      // Check command in Execution-Order-List available ?
      IF ( AxesGroup.Acyclic.ActiveCommandRegister.ExecutionOrderList[_listIdx] > EMPTY_EOL_ENTRY)
      THEN
        // set current SEQ / ACk index
        Telegram.PlcToRob.Sequence[_seqIdx].Header.SEQ_ACK := AxesGroup.State.CurrentSEQ[_seqIdx];
        
        // get active command register index
       _regIdx := AxesGroup.Acyclic.ActiveCommandRegister.ExecutionOrderList[_listIdx];
    
        // check State of the current ACR entry ?
        IF (( AxesGroup.Acyclic.ActiveCommandRegister.Register[_regIdx].Command[ACTIVE_CMD].State >= BufferStateCmd.CREATED  ) AND
            ( AxesGroup.Acyclic.ActiveCommandRegister.Register[_regIdx].Command[ACTIVE_CMD].State <= BufferStateCmd.SENDING  ))
        THEN
          // add size of fragement header      
          Telegram.PlcToRob.Sequence[_seqIdx].Header.PayloadLength :=
            Telegram.PlcToRob.Sequence[_seqIdx].Header.PayloadLength + SIZEOF(Telegram.PlcToRob.Sequence[_seqIdx].Fragment[_fragIdx].Header); 
            
            
          Telegram.PlcToRob.Sequence[_seqIdx].Fragment[_fragIdx].Header.CmdID          := AxesGroup.Acyclic.ActiveCommandRegister.Register[_regIdx].UniqueID;
          Telegram.PlcToRob.Sequence[_seqIdx].Fragment[_fragIdx].Header.Reserve        := 0;
          Telegram.PlcToRob.Sequence[_seqIdx].Fragment[_fragIdx].Header.FragmentAction := 0; // will be set below
          Telegram.PlcToRob.Sequence[_seqIdx].Fragment[_fragIdx].Header.PayloadPointer := AxesGroup.Acyclic.ActiveCommandRegister.Register[_regIdx].Command[ACTIVE_CMD].PayLoadPtr; 
          
          // The 1st message resets the ACR entry on the server side  
         _fragmentAction.Reset := (( AxesGroup.Acyclic.ActiveCommandRegister.Register[_regIdx].Command[ACTIVE_CMD].State      = BufferStateCmd.CREATED ) AND
                                   ( AxesGroup.Acyclic.ActiveCommandRegister.Register[_regIdx].Command[ACTIVE_CMD].PayLoadPtr = 0                      ));
                                   
          // Update messages must clear the ACR entry on the server side  
         _fragmentAction.Clear := (( AxesGroup.Acyclic.ActiveCommandRegister.Register[_regIdx].Command[ACTIVE_CMD].State      = BufferStateCmd.UPDATE_AVAILABLE  ) AND
                                   ( AxesGroup.Acyclic.ActiveCommandRegister.Register[_regIdx].Command[ACTIVE_CMD].PayLoadPtr = 0                                )); 
    
          
          // fill telegramm header - just for later debugging ( the header is part of the command payload itselfy ) {{{
          Telegram.PlcToRob.Sequence[_seqIdx].Fragment[_fragIdx].Command.Header.CmdType       := CombineBytesToUint ( AxesGroup.Acyclic.ActiveCommandRegister.Register[_regIdx].Command[ACTIVE_CMD].Payload[0],
                                                                                                                      AxesGroup.Acyclic.ActiveCommandRegister.Register[_regIdx].Command[ACTIVE_CMD].Payload[1]);
          Telegram.PlcToRob.Sequence[_seqIdx].Fragment[_fragIdx].Command.Header.ExecMode.0    :=                      AxesGroup.Acyclic.ActiveCommandRegister.Register[_regIdx].Command[ACTIVE_CMD].Payload[2].0;
          Telegram.PlcToRob.Sequence[_seqIdx].Fragment[_fragIdx].Command.Header.ExecMode.1    :=                      AxesGroup.Acyclic.ActiveCommandRegister.Register[_regIdx].Command[ACTIVE_CMD].Payload[2].1;
          Telegram.PlcToRob.Sequence[_seqIdx].Fragment[_fragIdx].Command.Header.ExecMode.2    :=                      AxesGroup.Acyclic.ActiveCommandRegister.Register[_regIdx].Command[ACTIVE_CMD].Payload[2].2;
          Telegram.PlcToRob.Sequence[_seqIdx].Fragment[_fragIdx].Command.Header.ExecMode.3    :=                      AxesGroup.Acyclic.ActiveCommandRegister.Register[_regIdx].Command[ACTIVE_CMD].Payload[2].3;
          Telegram.PlcToRob.Sequence[_seqIdx].Fragment[_fragIdx].Command.Header.Prio.0        :=                      AxesGroup.Acyclic.ActiveCommandRegister.Register[_regIdx].Command[ACTIVE_CMD].Payload[3].0;
          Telegram.PlcToRob.Sequence[_seqIdx].Fragment[_fragIdx].Command.Header.Prio.1        :=                      AxesGroup.Acyclic.ActiveCommandRegister.Register[_regIdx].Command[ACTIVE_CMD].Payload[3].1;
          Telegram.PlcToRob.Sequence[_seqIdx].Fragment[_fragIdx].Command.Header.Prio.2        :=                      AxesGroup.Acyclic.ActiveCommandRegister.Register[_regIdx].Command[ACTIVE_CMD].Payload[3].2;
          Telegram.PlcToRob.Sequence[_seqIdx].Fragment[_fragIdx].Command.Header.Prio.3        :=                      AxesGroup.Acyclic.ActiveCommandRegister.Register[_regIdx].Command[ACTIVE_CMD].Payload[3].3;
          Telegram.PlcToRob.Sequence[_seqIdx].Fragment[_fragIdx].Command.Header.ParSequence.0 :=                      AxesGroup.Acyclic.ActiveCommandRegister.Register[_regIdx].Command[ACTIVE_CMD].Payload[3].4;
          Telegram.PlcToRob.Sequence[_seqIdx].Fragment[_fragIdx].Command.Header.ParSequence.1 :=                      AxesGroup.Acyclic.ActiveCommandRegister.Register[_regIdx].Command[ACTIVE_CMD].Payload[3].5;
          Telegram.PlcToRob.Sequence[_seqIdx].Fragment[_fragIdx].Command.Header.ParSequence.2 :=                      AxesGroup.Acyclic.ActiveCommandRegister.Register[_regIdx].Command[ACTIVE_CMD].Payload[3].6;
          Telegram.PlcToRob.Sequence[_seqIdx].Fragment[_fragIdx].Command.Header.ParSequence.3 :=                      AxesGroup.Acyclic.ActiveCommandRegister.Register[_regIdx].Command[ACTIVE_CMD].Payload[3].7;
          // }}}
          // loop through the payload
          FOR _payLoadPtr := AxesGroup.Acyclic.ActiveCommandRegister.Register[_regIdx].Command[ACTIVE_CMD].PayLoadPtr TO AxesGroup.Acyclic.ActiveCommandRegister.Register[_regIdx].Command[ACTIVE_CMD].PayloadLen -1  
          DO
            // copy payload
            Telegram.PlcToRob.Sequence[_seqIdx].Fragment[_fragIdx].Command.Payload[_payLoadPtr] 
              := AxesGroup.Acyclic.ActiveCommandRegister.Register[_regIdx].Command[ACTIVE_CMD].Payload[_payLoadPtr];
        
            // inc current sequence payload length
            Telegram.PlcToRob.Sequence[_seqIdx].Header.PayloadLength
              := Telegram.PlcToRob.Sequence[_seqIdx].Header.PayloadLength + 1;  
        
            // inc current fragment payload length
            Telegram.PlcToRob.Sequence[_seqIdx].Fragment[_fragIdx].Header.PayloadLength 
              := Telegram.PlcToRob.Sequence[_seqIdx].Fragment[_fragIdx].Header.PayloadLength + 1;
        
            // inc payload pointer in active command register
            AxesGroup.Acyclic.ActiveCommandRegister.Register[_regIdx].Command[ACTIVE_CMD].PayLoadPtr 
              := AxesGroup.Acyclic.ActiveCommandRegister.Register[_regIdx].Command[ACTIVE_CMD].PayLoadPtr + 1;
          
            // set command state
            IF ( AxesGroup.Acyclic.ActiveCommandRegister.Register[_regIdx].Command[ACTIVE_CMD].PayLoadPtr >= AxesGroup.Acyclic.ActiveCommandRegister.Register[_regIdx].Command[ACTIVE_CMD].PayLoadLen) 
            THEN
              AxesGroup.Acyclic.ActiveCommandRegister.Register[_regIdx].Command[ACTIVE_CMD].State := BufferStateCmd.PROCESSED;
            ELSE
              AxesGroup.Acyclic.ActiveCommandRegister.Register[_regIdx].Command[ACTIVE_CMD].State := BufferStateCmd.SENDING;  
            END_IF 
    
            // calc current telegram payload length
           _telegramLengthCurrent := CalculateTelegramLengthPlcToRob(AxesGroup := AxesGroup);
      
            // check limit reached ?
            IF ( _telegramLengthCurrent >= _parCfg.Com.TelegramLengthPlcToRob) 
            THEN  
              EXIT; // -> abort for loop 
            END_IF  
          END_FOR
    
          // check payload complete ?
         _fragmentAction.Complete := AxesGroup.Acyclic.ActiveCommandRegister.Register[_regIdx].Command[ACTIVE_CMD].PayLoadPtr 
                                  >= AxesGroup.Acyclic.ActiveCommandRegister.Register[_regIdx].Command[ACTIVE_CMD].PayloadLen;
    
          // just for brakepoint
          IF (_fragmentAction.Complete)
          THEN
           _fragmentAction.Complete := _fragmentAction.Complete; 
          END_IF
    
          // set fragment action
          Telegram.PlcToRob.Sequence[_seqIdx].Fragment[_fragIdx].Header.FragmentAction := FragmentActionToByte(_fragmentAction);
        END_IF
      END_IF
      
      // inc execution order list index 
     _listIdx := _listIdx + 1;
      // inc fragment index 
     _fragIdx := _fragIdx + 1;
  
      // check abort conditions
      IF (( _telegramLengthCurrent                                                >= _parCfg.Com.TelegramLengthPlcToRob  ) OR  // Payload limit reached 
          ( _fragIdx                                                              >=  RobotLibraryParameter.FRAGMENT_MAX ) OR  // Max fragment limit reached
          (  AxesGroup.Acyclic.ActiveCommandRegister.ExecutionOrderList[_listIdx]  =  EMPTY_EOL_ENTRY                    ))    // No entry in ExecutionOrderList left
      THEN
        EXIT;// -> Abort while loop
      END_IF         
    END_WHILE  
    
    AxesGroup.State.SequenceCountSend          := _seqIdx;
    AxesGroup.State.FragmentCountSend[_seqIdx] := _fragIdx;
    
  END_IF  
END_FOR
                
END_METHOD

METHOD CalculateCyclicDataLength : UINT
VAR_IN_OUT
  /// Robot assignment of function
  AxesGroup : AxesGroup;
END_VAR
VAR_INPUT
  /// Communication direction
  Direction : ComDirection;
END_VAR

VAR CONSTANT
  /// Size of the header
  ROB_TO_PLC_HEADER_SIZE : UINT := 10;
END_VAR
                  // ------------------------------------
// PLC -> ROB
// ------------------------------------
IF (Direction = ComDirection.PLC_TO_ROB)
THEN  
  // Add Header size 
  CalculateCyclicDataLength := CalculateCyclicDataLength + SIZEOF(Telegram.PlcToRob.Header);  
  // Add Cyclic size 
  CalculateCyclicDataLength := CalculateCyclicDataLength + SIZEOF(Telegram.PlcToRob.Cyclic);
  
  // Check SubProgramData active ? 
  IF ( AxesGroup.CyclicOptional.PlcToRob.SubProgramData.Active )
  THEN
    // Add SubProgramData size 
    CalculateCyclicDataLength := CalculateCyclicDataLength + SIZEOF(Telegram.PlcToRob.CyclicOptional.SubProgramData);
  END_IF
    
  // Check CartesianPosition active ? 
  IF ( AxesGroup.CyclicOptional.PlcToRob.CartesianPosition.Active )
  THEN
    // Add CartesianPosition size 
    CalculateCyclicDataLength := CalculateCyclicDataLength + SIZEOF(Telegram.PlcToRob.CyclicOptional.CartesianPosition);
  END_IF
  
  // Check JointPosition active ? 
  IF ( AxesGroup.CyclicOptional.PlcToRob.JointPosition.Active )
  THEN
    // Add JointPosition size 
    CalculateCyclicDataLength := CalculateCyclicDataLength + SIZEOF(Telegram.PlcToRob.CyclicOptional.JointPosition);
  END_IF  
  
  // Check Force active ? 
  IF ( AxesGroup.CyclicOptional.PlcToRob.Force.Active )
  THEN
    // Add Force size 
    CalculateCyclicDataLength := CalculateCyclicDataLength + SIZEOF(Telegram.PlcToRob.CyclicOptional.Force);
  END_IF  
    
  // Check CartesianPositionExt acive ? 
  IF ( AxesGroup.CyclicOptional.PlcToRob.CartesianPositionExt.Active )
  THEN
    // Add CartesianPositionExt size 
    CalculateCyclicDataLength := CalculateCyclicDataLength + SIZEOF(Telegram.PlcToRob.CyclicOptional.CartesianPositionExt);
  END_IF   
    
  // Check JointPositionExt active ?
  IF ( AxesGroup.CyclicOptional.PlcToRob.JointPositionExt.Active )
  THEN
    // Add JointPositionExt size 
    CalculateCyclicDataLength := CalculateCyclicDataLength + SIZEOF(Telegram.PlcToRob.CyclicOptional.JointPositionExt);
  END_IF  
        
  // Check ForceExt active ?
  IF ( AxesGroup.CyclicOptional.PlcToRob.ForceExt.Active )
  THEN
    // Add ForceExt size 
    CalculateCyclicDataLength := CalculateCyclicDataLength + SIZEOF(Telegram.PlcToRob.CyclicOptional.ForceExt);
  END_IF
END_IF

// ------------------------------------
// ROB -> PLC
// ------------------------------------
IF (Direction = ComDirection.ROB_TO_PLC)
THEN
  // Add Header size 
  CalculateCyclicDataLength := CalculateCyclicDataLength + ROB_TO_PLC_HEADER_SIZE; 
  {warning 'ToDo: Used a constant because SizeOf(Telegram.RobToPlc.Header) return a wrong value,  because of VersionStruct instead of Byte'}
  
  // Check SubProgramData active ? 
  IF ( AxesGroup.CyclicOptional.RobToPlc.SubProgramData.Active )
  THEN
    // Add SubProgramData size 
    CalculateCyclicDataLength := CalculateCyclicDataLength + SIZEOF(Telegram.RobToPlc.CyclicOptional.SubProgramData);
  END_IF
    
  // Check CartesianPosition active ? 
  IF ( AxesGroup.CyclicOptional.RobToPlc.CartesianPosition.Active )
  THEN
    // Add CartesianPosition size 
    CalculateCyclicDataLength := CalculateCyclicDataLength + SIZEOF(Telegram.RobToPlc.CyclicOptional.CartesianPosition);
  END_IF
  
  // Check JointPosition active ? 
  IF ( AxesGroup.CyclicOptional.RobToPlc.JointPosition.Active )
  THEN
    // Add JointPosition size 
    CalculateCyclicDataLength := CalculateCyclicDataLength + SIZEOF(Telegram.RobToPlc.CyclicOptional.JointPosition);
  END_IF  
  
  // Check Force active ? 
  IF ( AxesGroup.CyclicOptional.RobToPlc.Force.Active )
  THEN
    // Add Force size 
    CalculateCyclicDataLength := CalculateCyclicDataLength + SIZEOF(Telegram.RobToPlc.CyclicOptional.Force);
  END_IF  
    
  // Check Current acive ? 
  IF ( AxesGroup.CyclicOptional.RobToPlc.Current.Active )
  THEN
    // Add Current size 
    CalculateCyclicDataLength := CalculateCyclicDataLength + SIZEOF(Telegram.RobToPlc.CyclicOptional.Current);
  END_IF    
    
  // Check CartesianPositionExt acive ? 
  IF ( AxesGroup.CyclicOptional.RobToPlc.CartesianPositionExt.Active )
  THEN
    // Add CartesianPositionExt size 
    CalculateCyclicDataLength := CalculateCyclicDataLength + SIZEOF(Telegram.RobToPlc.CyclicOptional.CartesianPositionExt);
  END_IF  
    
  // Check JointPositionExt active ?
  IF ( AxesGroup.CyclicOptional.RobToPlc.JointPositionExt.Active )
  THEN
    // Add JointPositionExt size 
    CalculateCyclicDataLength := CalculateCyclicDataLength + SIZEOF(Telegram.RobToPlc.CyclicOptional.JointPositionExt);
  END_IF  
        
  // Check ForceExt active ?
  IF ( AxesGroup.CyclicOptional.RobToPlc.ForceExt.Active )
  THEN
    // Add ForceExt size 
    CalculateCyclicDataLength := CalculateCyclicDataLength + SIZEOF(Telegram.RobToPlc.CyclicOptional.ForceExt);
  END_IF
    
  // Check CurrentExt active ? 
  IF ( AxesGroup.CyclicOptional.RobToPlc.CurrentExt.Active )
  THEN
    // Add CurrentExt size 
    CalculateCyclicDataLength := CalculateCyclicDataLength + SIZEOF(Telegram.RobToPlc.CyclicOptional.CurrentExt);
  END_IF
END_IF
                
END_METHOD

METHOD CalculateSequencePayloadMax : UINT
VAR_IN_OUT
  /// Robot assignment of function
  AxesGroup : AxesGroup;
END_VAR
VAR_INPUT
  /// Communication direction
  Direction : ComDirection;
  /// Sequeunce
  Sequence : SequenceFlag;  
END_VAR

VAR
  /// Length of the cyclic header
 _cyclicDataLength      : UINT;
END_VAR
                  // calculate cyclic header length
_cyclicDataLength := CalculateCyclicDataLength(AxesGroup := AxesGroup, Direction := Direction);


CASE (Sequence) 
OF
  SequenceFlag.PRIMARY_SEQUENCE   : 

    IF (Direction = ComDirection.PLC_TO_ROB)
    THEN  
      // calculate sequence payload length
      CalculateSequencePayloadMax := ( _parCfg.Com.TelegramLengthPlcToRob - _cyclicDataLength );
    END_IF

